LIN {X 0,Y 222.281,Z 512.285,A -85,B 0,C 180,E1 -22174.841,E2 -22174.841} C_VEL
LIN {X 0,Y 219.936,Z 524.701,A -85,B 0,C 180,E1 -22175.823,E2 -22175.823} C_VEL
LIN {X 0,Y 217.033,Z 536.462,A -85,B 0,C 180,E1 -22177.118,E2 -22177.118} C_VEL
LIN {X 0,Y 213.717,Z 547.223,A -85,B 0,C 180,E1 -22178.669,E2 -22178.669} C_VEL
LIN {X 0,Y 209.672,Z 558.118,A -85,B 0,C 180,E1 -22180.681,E2 -22180.681} C_VEL
LIN {X 0,Y 206.055,Z 566.605,A -85,B 0,C 180,E1 -22182.687,E2 -22182.687} C_VEL
LIN {X 0,Y 201.983,Z 575.031,A -85,B 0,C 180,E1 -22185.204,E2 -22185.204} C_VEL
LIN {X 0,Y 197.556,Z 583.105,A -85,B 0,C 180,E1 -22188.338,E2 -22188.338} C_VEL
LIN {X 0,Y 193.488,Z 589.856,A -85,B 0,C 180,E1 -22191.868,E2 -22191.868} C_VEL
LIN {X 0,Y 190.43,Z 594.406,A -85,B 0,C 180,E1 -22195.108,E2 -22195.108} C_VEL
LIN {X 0,Y 187.913,Z 597.772,A -85,B 0,C 180,E1 -22198.426,E2 -22198.426} C_VEL
LIN {X 0,Y 186.57,Z 599.41,A -85,B 0,C 180,E1 -22200.68,E2 -22200.68} C_VEL
LIN {X 0,Y 185.448,Z 600.607,A -85,B 0,C 180,E1 -22202.951,E2 -22202.951} C_VEL
LIN {X 0,Y 184.224,Z 601.526,A -85,B 0,C 180,E1 -22206.29,E2 -22206.29} C_VEL
LIN {X 0,Y 183.363,Z 601.506,A -85,B 0,C 180,E1 -22209.821,E2 -22209.821} C_VEL
LIN {X 0,Y 183.025,Z 600.3,A -85,B 0,C 180,E1 -22213.738,E2 -22213.738} C_VEL
LIN {X 0,Y 183.035,Z 598.555,A -85,B 0,C 180,E1 -22216.681,E2 -22216.681} C_VEL
LIN {X 0,Y 183.469,Z 595.61,A -85,B 0,C 180,E1 -22220.074,E2 -22220.074} C_VEL
LIN {X 0,Y 184.219,Z 591.613,A -85,B 0,C 180,E1 -22223.428,E2 -22223.428} C_VEL
LIN {X 0,Y 185.498,Z 585.472,A -85,B 0,C 180,E1 -22227.286,E2 -22227.286} C_VEL
LIN {X 0,Y 186.993,Z 578.75,A -85,B 0,C 180,E1 -22230.538,E2 -22230.538} C_VEL
LIN {X 0,Y 189.001,Z 570.397,A -85,B 0,C 180,E1 -22233.731,E2 -22233.731} C_VEL
LIN {X 0,Y 191.015,Z 561.82,A -85,B 0,C 180,E1 -22236.337,E2 -22236.337} C_VEL
LIN {X 0,Y 193.269,Z 551.234,A -85,B 0,C 180,E1 -22238.89,E2 -22238.89} C_VEL
LIN {X 0,Y 195.356,Z 540.725,A -85,B 0,C 180,E1 -22240.887,E2 -22240.887} C_VEL
LIN {X 0,Y 197.304,Z 529.166,A -85,B 0,C 180,E1 -22242.601,E2 -22242.601} C_VEL
LIN {X 0,Y 198.932,Z 517.169,A -85,B 0,C 180,E1 -22243.926,E2 -22243.926} C_VEL
LIN {X 0,Y 200.159,Z 504.209,A -85,B 0,C 180,E1 -22244.947,E2 -22244.947} C_VEL
LIN {X 0,Y 200.893,Z 491.969,A -85,B 0,C 180,E1 -22245.549,E2 -22245.549} C_VEL
LIN {X 0,Y 203.334,Z 436.009,A -85,B 0,C 180,E1 -22247.426,E2 -22247.426} C_VEL
LIN {X 0,Y 199.401,Z 426.13,A -85,B 0,C 180,E1 -22248.427,E2 -22248.427} C_VEL
LIN {X 0,Y 192.691,Z 412.029,A -85,B 0,C 180,E1 -22250.125,E2 -22250.125} C_VEL
LIN {X 0,Y 186.668,Z 401.306,A -85,B 0,C 180,E1 -22251.692,E2 -22251.692} C_VEL
LIN {X 0,Y 185.603,Z 398.365,A -85,B 0,C 180,E1 -22252.033,E2 -22252.033} C_VEL
LIN {X 0,Y 185.566,Z 398.373,A -85,B 0,C 180,E1 -22257.031,E2 -22257.031} C_VEL
LIN {X 0,Y 185.581,Z 398.368,A -85,B 0,C 180,E1 -22259.492,E2 -22259.492} C_VEL
LIN {X 0,Y 185.501,Z 398.379,A -85,B 0,C 180,E1 -22264.631,E2 -22264.631} C_VEL
LIN {X 0,Y 185.506,Z 398.373,A -85,B 0,C 180,E1 -22267.312,E2 -22267.312} C_VEL
LIN {X 0,Y 185.472,Z 398.376,A -85,B 0,C 180,E1 -22270.724,E2 -22270.724} C_VEL
LIN {X 0,Y 185.461,Z 398.376,A -85,B 0,C 180,E1 -22276.053,E2 -22276.053} C_VEL
LIN {X 0,Y 185.468,Z 398.38,A -85,B 0,C 180,E1 -22279.894,E2 -22279.894} C_VEL
LIN {X 0,Y 185.505,Z 398.369,A -85,B 0,C 180,E1 -22282.71,E2 -22282.71} C_VEL
LIN {X 0,Y 185.541,Z 398.369,A -85,B 0,C 180,E1 -22287.974,E2 -22287.974} C_VEL
LIN {X 0,Y 185.58,Z 398.361,A -85,B 0,C 180,E1 -22290.575,E2 -22290.575} C_VEL
LIN {X 0,Y 185.585,Z 398.36,A -85,B 0,C 180,E1 -22295.381,E2 -22295.381} C_VEL
LIN {X 0,Y 185.672,Z 398.353,A -85,B 0,C 180,E1 -22301.132,E2 -22301.132} C_VEL
LIN {X 0,Y 185.692,Z 398.345,A -85,B 0,C 180,E1 -22304.636,E2 -22304.636} C_VEL
LIN {X 0,Y 185.886,Z 398.322,A -85,B 0,C 180,E1 -22309.417,E2 -22309.417} C_VEL
LIN {X 0,Y 185.948,Z 398.319,A -85,B 0,C 180,E1 -22313.489,E2 -22313.489} C_VEL
LIN {X 0,Y 186.203,Z 398.276,A -85,B 0,C 180,E1 -22317.836,E2 -22317.836} C_VEL
LIN {X 0,Y 186.402,Z 398.23,A -85,B 0,C 180,E1 -22319.999,E2 -22319.999} C_VEL
LIN {X 0,Y 185.914,Z 398.307,A -85,B 0,C 180,E1 -22324.335,E2 -22324.335} C_VEL
LIN {X 0,Y 185.979,Z 398.318,A -85,B 0,C 180,E1 -22328.693,E2 -22328.693} C_VEL
LIN {X 0,Y 185.725,Z 398.347,A -85,B 0,C 180,E1 -22333.123,E2 -22333.123} C_VEL
LIN {X 0,Y 185.686,Z 398.349,A -85,B 0,C 180,E1 -22337.625,E2 -22337.625} C_VEL
LIN {X 0,Y 185.593,Z 398.365,A -85,B 0,C 180,E1 -22342.251,E2 -22342.251} C_VEL
LIN {X 0,Y 185.559,Z 398.369,A -85,B 0,C 180,E1 -22347.032,E2 -22347.032} C_VEL
LIN {X 0,Y 185.576,Z 398.37,A -85,B 0,C 180,E1 -22349.493,E2 -22349.493} C_VEL
LIN {X 0,Y 185.518,Z 398.38,A -85,B 0,C 180,E1 -22354.628,E2 -22354.628} C_VEL
LIN {X 0,Y 185.565,Z 398.375,A -85,B 0,C 180,E1 -22357.314,E2 -22357.314} C_VEL
LIN {X 0,Y 185.559,Z 398.377,A -85,B 0,C 180,E1 -22360.758,E2 -22360.758} C_VEL
LIN {X 0,Y 185.562,Z 398.375,A -85,B 0,C 180,E1 -22366.022,E2 -22366.022} C_VEL
LIN {X 0,Y 185.597,Z 398.469,A -85,B 0,C 180,E1 -22368.091,E2 -22368.091} C_VEL
LIN {X 0,Y 187.363,Z 405.749,A -85,B 0,C 180,E1 -22371.972,E2 -22371.972} C_VEL
LIN {X 0,Y 193.883,Z 421.299,A -85,B 0,C 180,E1 -22373.81,E2 -22373.81} C_VEL
LIN {X 0,Y 199.191,Z 435.84,A -85,B 0,C 180,E1 -22375.277,E2 -22375.277} C_VEL
LIN {X 0,Y 202.246,Z 467.615,A -85,B 0,C 180,E1 -22377.009,E2 -22377.009} C_VEL
LIN {X 0,Y 201.243,Z 492.996,A -85,B 0,C 180,E1 -22377.874,E2 -22377.874} C_VEL
LIN {X 0,Y 200.356,Z 498.833,A -85,B 0,C 180,E1 -22377.976,E2 -22377.976} C_VEL
LIN {X 0,Y 194.089,Z 517.66,A -85,B 0,C 180,E1 -22377.992,E2 -22377.992} C_VEL
LIN {X 0,Y 193.08,Z 523.397,A -85,B 0,C 180,E1 -22378.283,E2 -22378.283} C_VEL
LIN {X 0,Y 191.502,Z 536.392,A -85,B 0,C 180,E1 -22379.39,E2 -22379.39} C_VEL
LIN {X 0,Y 189.488,Z 548.643,A -85,B 0,C 180,E1 -22380.87,E2 -22380.87} C_VEL
LIN {X 0,Y 187.158,Z 559.674,A -85,B 0,C 180,E1 -22382.613,E2 -22382.613} C_VEL
LIN {X 0,Y 184.678,Z 570.968,A -85,B 0,C 180,E1 -22384.953,E2 -22384.953} C_VEL
LIN {X 0,Y 182.546,Z 580.085,A -85,B 0,C 180,E1 -22387.357,E2 -22387.357} C_VEL
LIN {X 0,Y 181.162,Z 585.57,A -85,B 0,C 180,E1 -22389.077,E2 -22389.077} C_VEL
LIN {X 0,Y 179.534,Z 592.745,A -85,B 0,C 180,E1 -22391.75,E2 -22391.75} C_VEL
LIN {X 0,Y 177.925,Z 600.065,A -85,B 0,C 180,E1 -22395.123,E2 -22395.123} C_VEL
LIN {X 0,Y 176.898,Z 605.891,A -85,B 0,C 180,E1 -22398.542,E2 -22398.542} C_VEL
LIN {X 0,Y 176.379,Z 610.455,A -85,B 0,C 180,E1 -22401.984,E2 -22401.984} C_VEL
LIN {X 0,Y 176.174,Z 614.18,A -85,B 0,C 180,E1 -22405.792,E2 -22405.792} C_VEL
LIN {X 0,Y 176.394,Z 616.866,A -85,B 0,C 180,E1 -22410,E2 -22410} C_VEL
LIN {X 0,Y 176.156,Z 618.092,A -85,B 0,C 180,E1 -22414.128,E2 -22414.128} C_VEL
LIN {X 0,Y 176.21,Z 618.167,A -85,B 0,C 180,E1 -22416.872,E2 -22416.872} C_VEL
LIN {X 0,Y 176.95,Z 617.068,A -85,B 0,C 180,E1 -22421.454,E2 -22421.454} C_VEL
LIN {X 0,Y 177.682,Z 615.947,A -85,B 0,C 180,E1 -22423.728,E2 -22423.728} C_VEL
LIN {X 0,Y 178.687,Z 614.389,A -85,B 0,C 180,E1 -22425.981,E2 -22425.981} C_VEL
LIN {X 0,Y 180.91,Z 611.301,A -85,B 0,C 180,E1 -22429.281,E2 -22429.281} C_VEL
LIN {X 0,Y 183.636,Z 607.189,A -85,B 0,C 180,E1 -22432.501,E2 -22432.501} C_VEL
LIN {X 0,Y 187.434,Z 600.937,A -85,B 0,C 180,E1 -22436.139,E2 -22436.139} C_VEL
LIN {X 0,Y 191.356,Z 594.172,A -85,B 0,C 180,E1 -22439.119,E2 -22439.119} C_VEL
LIN {X 0,Y 195.968,Z 585.811,A -85,B 0,C 180,E1 -22441.936,E2 -22441.936} C_VEL
LIN {X 0,Y 200.127,Z 577.24,A -85,B 0,C 180,E1 -22444.185,E2 -22444.185} C_VEL
LIN {X 0,Y 204.678,Z 566.714,A -85,B 0,C 180,E1 -22446.32,E2 -22446.32} C_VEL
LIN {X 0,Y 208.619,Z 556.305,A -85,B 0,C 180,E1 -22447.937,E2 -22447.937} C_VEL
LIN {X 0,Y 212.179,Z 544.891,A -85,B 0,C 180,E1 -22449.306,E2 -22449.306} C_VEL
LIN {X 0,Y 215.33,Z 531.845,A -85,B 0,C 180,E1 -22450.441,E2 -22450.441} C_VEL
LIN {X 0,Y 217.654,Z 518.383,A -85,B 0,C 180,E1 -22451.247,E2 -22451.247} C_VEL
LIN {X 0,Y 218.894,Z 505.408,A -85,B 0,C 180,E1 -22451.736,E2 -22451.736} C_VEL
LIN {X 0,Y 220.857,Z 474.587,A -85,B 0,C 180,E1 -22452.675,E2 -22452.675} C_VEL
LIN {X 0,Y 220.319,Z 470.267,A -85,B 0,C 180,E1 -22453.05,E2 -22453.05} C_VEL
LIN {X 0,Y 215.13,Z 457.835,A -85,B 0,C 180,E1 -22455.335,E2 -22455.335} C_VEL
LIN {X 0,Y 209.768,Z 446.74,A -85,B 0,C 180,E1 -22457.874,E2 -22457.874} C_VEL
LIN {X 0,Y 204.194,Z 436.795,A -85,B 0,C 180,E1 -22460.756,E2 -22460.756} C_VEL
LIN {X 0,Y 201.189,Z 431.731,A -85,B 0,C 180,E1 -22462.459,E2 -22462.459} C_VEL
LIN {X 0,Y 197.894,Z 426.511,A -85,B 0,C 180,E1 -22464.466,E2 -22464.466} C_VEL
LIN {X 0,Y 194.017,Z 420.666,A -85,B 0,C 180,E1 -22467.088,E2 -22467.088} C_VEL
LIN {X 0,Y 190.602,Z 415.814,A -85,B 0,C 180,E1 -22469.73,E2 -22469.73} C_VEL
LIN {X 0,Y 189.536,Z 414.282,A -85,B 0,C 180,E1 -22470.639,E2 -22470.639} C_VEL
LIN {X 0,Y 185.502,Z 408.804,A -85,B 0,C 180,E1 -22474.537,E2 -22474.537} C_VEL
LIN {X 0,Y 184.714,Z 407.543,A -85,B 0,C 180,E1 -22475.441,E2 -22475.441} C_VEL
LIN {X 0,Y 181.501,Z 404.142,A -85,B 0,C 180,E1 -22479.605,E2 -22479.605} C_VEL
LIN {X 0,Y 179.041,Z 400.824,A -85,B 0,C 180,E1 -22484.49,E2 -22484.49} C_VEL
LIN {X 0,Y 178.646,Z 399.226,A -85,B 0,C 180,E1 -22486.202,E2 -22486.202} C_VEL
LIN {X 0,Y 178.955,Z 399.184,A -85,B 0,C 180,E1 -22490.963,E2 -22490.963} C_VEL
LIN {X 0,Y 179.15,Z 399.152,A -85,B 0,C 180,E1 -22497.752,E2 -22497.752} C_VEL
LIN {X 0,Y 179.315,Z 399.229,A -85,B 0,C 180,E1 -22500.351,E2 -22500.351} C_VEL
LIN {X 0,Y 179.788,Z 401.258,A -85,B 0,C 180,E1 -22501.821,E2 -22501.821} C_VEL
LIN {X 0,Y 181.116,Z 403.543,A -85,B 0,C 180,E1 -22504.452,E2 -22504.452} C_VEL
LIN {X 0,Y 184.311,Z 405.474,A -85,B 0,C 180,E1 -22508.567,E2 -22508.567} C_VEL
LIN {X 0,Y 185.791,Z 408.533,A -85,B 0,C 180,E1 -22510.377,E2 -22510.377} C_VEL
LIN {X 0,Y 188.224,Z 410.668,A -85,B 0,C 180,E1 -22512.672,E2 -22512.672} C_VEL
LIN {X 0,Y 188.96,Z 411.267,A -85,B 0,C 180,E1 -22513.306,E2 -22513.306} C_VEL
LIN {X 0,Y 190.801,Z 414.301,A -85,B 0,C 180,E1 -22514.943,E2 -22514.943} C_VEL
LIN {X 0,Y 193.337,Z 416.734,A -85,B 0,C 180,E1 -22516.839,E2 -22516.839} C_VEL
LIN {X 0,Y 195.579,Z 420.044,A -85,B 0,C 180,E1 -22518.465,E2 -22518.465} C_VEL
LIN {X 0,Y 197.368,Z 422.01,A -85,B 0,C 180,E1 -22519.604,E2 -22519.604} C_VEL
LIN {X 0,Y 200.297,Z 425.823,A -85,B 0,C 180,E1 -22521.385,E2 -22521.385} C_VEL
LIN {X 0,Y 204.844,Z 432.293,A -85,B 0,C 180,E1 -22523.921,E2 -22523.921} C_VEL
LIN {X 0,Y 209.465,Z 439.033,A -85,B 0,C 180,E1 -22526.238,E2 -22526.238} C_VEL
LIN {X 0,Y 215.672,Z 449.023,A -85,B 0,C 180,E1 -22529.062,E2 -22529.062} C_VEL
LIN {X 0,Y 219.882,Z 456.772,A -85,B 0,C 180,E1 -22530.825,E2 -22530.825} C_VEL
LIN {X 0,Y 221.735,Z 460.811,A -85,B 0,C 180,E1 -22531.591,E2 -22531.591} C_VEL
LIN {X 0,Y 219.07,Z 499.801,A -85,B 0,C 180,E1 -22532.809,E2 -22532.809} C_VEL
LIN {X 0,Y 217.235,Z 513.449,A -85,B 0,C 180,E1 -22533.56,E2 -22533.56} C_VEL
LIN {X 0,Y 214.826,Z 525.527,A -85,B 0,C 180,E1 -22534.54,E2 -22534.54} C_VEL
LIN {X 0,Y 211.585,Z 537.865,A -85,B 0,C 180,E1 -22535.941,E2 -22535.941} C_VEL
LIN {X 0,Y 207.934,Z 549.072,A -85,B 0,C 180,E1 -22537.626,E2 -22537.626} C_VEL
LIN {X 0,Y 203.941,Z 559.145,A -85,B 0,C 180,E1 -22539.552,E2 -22539.552} C_VEL
LIN {X 0,Y 199.411,Z 569.061,A -85,B 0,C 180,E1 -22542.04,E2 -22542.04} C_VEL
LIN {X 0,Y 195.133,Z 577.215,A -85,B 0,C 180,E1 -22544.659,E2 -22544.659} C_VEL
LIN {X 0,Y 190.814,Z 584.63,A -85,B 0,C 180,E1 -22547.758,E2 -22547.758} C_VEL
LIN {X 0,Y 187.617,Z 589.599,A -85,B 0,C 180,E1 -22550.447,E2 -22550.447} C_VEL
LIN {X 0,Y 184.211,Z 594.421,A -85,B 0,C 180,E1 -22553.872,E2 -22553.872} C_VEL
LIN {X 0,Y 181.551,Z 597.797,A -85,B 0,C 180,E1 -22557.184,E2 -22557.184} C_VEL
LIN {X 0,Y 180.078,Z 599.495,A -85,B 0,C 180,E1 -22559.513,E2 -22559.513} C_VEL
LIN {X 0,Y 178.792,Z 600.76,A -85,B 0,C 180,E1 -22561.856,E2 -22561.856} C_VEL
LIN {X 0,Y 177.277,Z 601.87,A -85,B 0,C 180,E1 -22565.76,E2 -22565.76} C_VEL
LIN {X 0,Y 176.405,Z 601.882,A -85,B 0,C 180,E1 -22568.989,E2 -22568.989} C_VEL
LIN {X 0,Y 176.063,Z 601.421,A -85,B 0,C 180,E1 -22571.377,E2 -22571.377} C_VEL
LIN {X 0,Y 175.949,Z 600.495,A -85,B 0,C 180,E1 -22573.764,E2 -22573.764} C_VEL
LIN {X 0,Y 175.927,Z 599.158,A -85,B 0,C 180,E1 -22576.132,E2 -22576.132} C_VEL
LIN {X 0,Y 176.282,Z 596.333,A -85,B 0,C 180,E1 -22579.665,E2 -22579.665} C_VEL
LIN {X 0,Y 177.051,Z 592.457,A -85,B 0,C 180,E1 -22583.161,E2 -22583.161} C_VEL
LIN {X 0,Y 178.082,Z 587.45,A -85,B 0,C 180,E1 -22586.606,E2 -22586.606} C_VEL
LIN {X 0,Y 179.517,Z 581.158,A -85,B 0,C 180,E1 -22590,E2 -22590} C_VEL
LIN {X 0,Y 181.476,Z 573.284,A -85,B 0,C 180,E1 -22593.33,E2 -22593.33} C_VEL
LIN {X 0,Y 183.442,Z 565.238,A -85,B 0,C 180,E1 -22596.048,E2 -22596.048} C_VEL
LIN {X 0,Y 185.817,Z 555.399,A -85,B 0,C 180,E1 -22598.701,E2 -22598.701} C_VEL
LIN {X 0,Y 187.782,Z 545.805,A -85,B 0,C 180,E1 -22600.785,E2 -22600.785} C_VEL
LIN {X 0,Y 189.817,Z 535.446,A -85,B 0,C 180,E1 -22602.563,E2 -22602.563} C_VEL
LIN {X 0,Y 191.722,Z 523.136,A -85,B 0,C 180,E1 -22604.19,E2 -22604.19} C_VEL
LIN {X 0,Y 193.209,Z 510.227,A -85,B 0,C 180,E1 -22605.426,E2 -22605.426} C_VEL
LIN {X 0,Y 194.24,Z 497.73,A -85,B 0,C 180,E1 -22606.217,E2 -22606.217} C_VEL
LIN {X 0,Y 197.004,Z 437.596,A -85,B 0,C 180,E1 -22608.331,E2 -22608.331} C_VEL
LIN {X 0,Y 191.815,Z 425.138,A -85,B 0,C 180,E1 -22609.712,E2 -22609.712} C_VEL
LIN {X 0,Y 185.069,Z 411.727,A -85,B 0,C 180,E1 -22611.523,E2 -22611.523} C_VEL
LIN {X 0,Y 179.955,Z 402.686,A -85,B 0,C 180,E1 -22612.96,E2 -22612.96} C_VEL
LIN {X 0,Y 178.668,Z 400,A -85,B 0,C 180,E1 -22613.357,E2 -22613.357} C_VEL
LIN {X 0,Y 178.523,Z 399.234,A -85,B 0,C 180,E1 -22613.484,E2 -22613.484} C_VEL
LIN {X 0,Y 178.49,Z 399.251,A -85,B 0,C 180,E1 -22618.196,E2 -22618.196} C_VEL
LIN {X 0,Y 178.503,Z 399.253,A -85,B 0,C 180,E1 -22620.785,E2 -22620.785} C_VEL
LIN {X 0,Y 178.487,Z 399.252,A -85,B 0,C 180,E1 -22624.218,E2 -22624.218} C_VEL
LIN {X 0,Y 178.396,Z 399.264,A -85,B 0,C 180,E1 -22629.073,E2 -22629.073} C_VEL
LIN {X 0,Y 178.399,Z 399.255,A -85,B 0,C 180,E1 -22632.044,E2 -22632.044} C_VEL
LIN {X 0,Y 178.395,Z 399.259,A -85,B 0,C 180,E1 -22635.162,E2 -22635.162} C_VEL
LIN {X 0,Y 178.403,Z 399.257,A -85,B 0,C 180,E1 -22638.458,E2 -22638.458} C_VEL
LIN {X 0,Y 178.421,Z 399.254,A -85,B 0,C 180,E1 -22643.782,E2 -22643.782} C_VEL
LIN {X 0,Y 178.484,Z 399.253,A -85,B 0,C 180,E1 -22646.545,E2 -22646.545} C_VEL
LIN {X 0,Y 178.521,Z 399.239,A -85,B 0,C 180,E1 -22650.006,E2 -22650.006} C_VEL
LIN {X 0,Y 178.523,Z 399.241,A -85,B 0,C 180,E1 -22654.882,E2 -22654.882} C_VEL
LIN {X 0,Y 178.621,Z 399.233,A -85,B 0,C 180,E1 -22660.783,E2 -22660.783} C_VEL
LIN {X 0,Y 178.654,Z 399.228,A -85,B 0,C 180,E1 -22666.347,E2 -22666.347} C_VEL
LIN {X 0,Y 178.911,Z 399.187,A -85,B 0,C 180,E1 -22670.959,E2 -22670.959} C_VEL
LIN {X 0,Y 178.866,Z 399.201,A -85,B 0,C 180,E1 -22675.492,E2 -22675.492} C_VEL
LIN {X 0,Y 179.366,Z 399.105,A -85,B 0,C 180,E1 -22679.999,E2 -22679.999} C_VEL
LIN {X 0,Y 178.862,Z 399.185,A -85,B 0,C 180,E1 -22684.507,E2 -22684.507} C_VEL
LIN {X 0,Y 178.907,Z 399.198,A -85,B 0,C 180,E1 -22689.04,E2 -22689.04} C_VEL
LIN {X 0,Y 178.653,Z 399.228,A -85,B 0,C 180,E1 -22693.652,E2 -22693.652} C_VEL
LIN {X 0,Y 178.62,Z 399.232,A -85,B 0,C 180,E1 -22699.216,E2 -22699.216} C_VEL
LIN {X 0,Y 178.531,Z 399.246,A -85,B 0,C 180,E1 -22705.124,E2 -22705.124} C_VEL
LIN {X 0,Y 178.476,Z 399.255,A -85,B 0,C 180,E1 -22710.791,E2 -22710.791} C_VEL
LIN {X 0,Y 178.482,Z 399.258,A -85,B 0,C 180,E1 -22714.22,E2 -22714.22} C_VEL
LIN {X 0,Y 178.47,Z 399.26,A -85,B 0,C 180,E1 -22719.055,E2 -22719.055} C_VEL
LIN {X 0,Y 178.497,Z 399.258,A -85,B 0,C 180,E1 -22722.016,E2 -22722.016} C_VEL
LIN {X 0,Y 178.529,Z 399.317,A -85,B 0,C 180,E1 -22727.116,E2 -22727.116} C_VEL
LIN {X 0,Y 180.026,Z 405.349,A -85,B 0,C 180,E1 -22730.522,E2 -22730.522} C_VEL
LIN {X 0,Y 187.418,Z 422.385,A -85,B 0,C 180,E1 -22732.724,E2 -22732.724} C_VEL
LIN {X 0,Y 193.121,Z 437.955,A -85,B 0,C 180,E1 -22734.391,E2 -22734.391} C_VEL
LIN {X 0,Y 195.928,Z 467.915,A -85,B 0,C 180,E1 -22736.091,E2 -22736.091} C_VEL
LIN {X 0,Y 193.825,Z 514.316,A -85,B 0,C 180,E1 -22737.745,E2 -22737.745} C_VEL
LIN {X 0,Y 193.08,Z 523.397,A -85,B 0,C 180,E1 -22738.283,E2 -22738.283} C_VEL
LIN {X 0,Y 191.912,Z 529.074,A -85,B 0,C 180,E1 -22738.622,E2 -22738.622} C_VEL
LIN {X 0,Y 188.076,Z 538.074,A -85,B 0,C 180,E1 -22739.117,E2 -22739.117} C_VEL
LIN {X 0,Y 183.906,Z 546.775,A -85,B 0,C 180,E1 -22739.846,E2 -22739.846} C_VEL
LIN {X 0,Y 182.235,Z 551.985,A -85,B 0,C 180,E1 -22740.551,E2 -22740.551} C_VEL
LIN {X 0,Y 179.822,Z 562.227,A -85,B 0,C 180,E1 -22742.348,E2 -22742.348} C_VEL
LIN {X 0,Y 177.947,Z 570.778,A -85,B 0,C 180,E1 -22744.251,E2 -22744.251} C_VEL
LIN {X 0,Y 175.612,Z 580.306,A -85,B 0,C 180,E1 -22746.872,E2 -22746.872} C_VEL
LIN {X 0,Y 174.172,Z 585.886,A -85,B 0,C 180,E1 -22748.706,E2 -22748.706} C_VEL
LIN {X 0,Y 172.171,Z 594.492,A -85,B 0,C 180,E1 -22752.173,E2 -22752.173} C_VEL
LIN {X 0,Y 170.54,Z 601.357,A -85,B 0,C 180,E1 -22755.685,E2 -22755.685} C_VEL
LIN {X 0,Y 169.653,Z 606.846,A -85,B 0,C 180,E1 -22759.257,E2 -22759.257} C_VEL
LIN {X 0,Y 169.237,Z 611.11,A -85,B 0,C 180,E1 -22762.844,E2 -22762.844} C_VEL
LIN {X 0,Y 169.088,Z 613.927,A -85,B 0,C 180,E1 -22765.978,E2 -22765.978} C_VEL
LIN {X 0,Y 169.31,Z 616.411,A -85,B 0,C 180,E1 -22770,E2 -22770} C_VEL
LIN {X 0,Y 169.078,Z 617.648,A -85,B 0,C 180,E1 -22773.976,E2 -22773.976} C_VEL
LIN {X 0,Y 169.139,Z 617.848,A -85,B 0,C 180,E1 -22777.161,E2 -22777.161} C_VEL
LIN {X 0,Y 169.976,Z 616.818,A -85,B 0,C 180,E1 -22781.931,E2 -22781.931} C_VEL
LIN {X 0,Y 170.747,Z 615.737,A -85,B 0,C 180,E1 -22784.297,E2 -22784.297} C_VEL
LIN {X 0,Y 171.852,Z 614.247,A -85,B 0,C 180,E1 -22786.634,E2 -22786.634} C_VEL
LIN {X 0,Y 174.207,Z 611.227,A -85,B 0,C 180,E1 -22790.054,E2 -22790.054} C_VEL
LIN {X 0,Y 177.093,Z 607.188,A -85,B 0,C 180,E1 -22793.381,E2 -22793.381} C_VEL
LIN {X 0,Y 181.079,Z 601.037,A -85,B 0,C 180,E1 -22797.13,E2 -22797.13} C_VEL
LIN {X 0,Y 185.181,Z 594.375,A -85,B 0,C 180,E1 -22800.189,E2 -22800.189} C_VEL
LIN {X 0,Y 190.003,Z 586.143,A -85,B 0,C 180,E1 -22803.064,E2 -22803.064} C_VEL
LIN {X 0,Y 194.327,Z 577.753,A -85,B 0,C 180,E1 -22805.355,E2 -22805.355} C_VEL
LIN {X 0,Y 199.035,Z 567.432,A -85,B 0,C 180,E1 -22807.524,E2 -22807.524} C_VEL
LIN {X 0,Y 203.627,Z 555.83,A -85,B 0,C 180,E1 -22809.359,E2 -22809.359} C_VEL
LIN {X 0,Y 207.332,Z 544.367,A -85,B 0,C 180,E1 -22810.731,E2 -22810.731} C_VEL
LIN {X 0,Y 210.583,Z 531.259,A -85,B 0,C 180,E1 -22811.872,E2 -22811.872} C_VEL
LIN {X 0,Y 212.824,Z 518.755,A -85,B 0,C 180,E1 -22812.625,E2 -22812.625} C_VEL
LIN {X 0,Y 214.188,Z 505.476,A -85,B 0,C 180,E1 -22813.141,E2 -22813.141} C_VEL
LIN {X 0,Y 216.16,Z 475.771,A -85,B 0,C 180,E1 -22814.055,E2 -22814.055} C_VEL
LIN {X 0,Y 215.814,Z 473.339,A -85,B 0,C 180,E1 -22814.292,E2 -22814.292} C_VEL
LIN {X 0,Y 210.516,Z 460.485,A -85,B 0,C 180,E1 -22816.799,E2 -22816.799} C_VEL
LIN {X 0,Y 206.06,Z 451.173,A -85,B 0,C 180,E1 -22819.062,E2 -22819.062} C_VEL
LIN {X 0,Y 200.931,Z 441.751,A -85,B 0,C 180,E1 -22821.891,E2 -22821.891} C_VEL
LIN {X 0,Y 198.036,Z 436.799,A -85,B 0,C 180,E1 -22823.637,E2 -22823.637} C_VEL
LIN {X 0,Y 195.352,Z 432.363,A -85,B 0,C 180,E1 -22825.379,E2 -22825.379} C_VEL
LIN {X 0,Y 191.747,Z 426.753,A -85,B 0,C 180,E1 -22827.974,E2 -22827.974} C_VEL
LIN {X 0,Y 188.425,Z 421.719,A -85,B 0,C 180,E1 -22830.723,E2 -22830.723} C_VEL
LIN {X 0,Y 183.755,Z 415.061,A -85,B 0,C 180,E1 -22835.422,E2 -22835.422} C_VEL
LIN {X 0,Y 183.077,Z 414.113,A -85,B 0,C 180,E1 -22836.23,E2 -22836.23} C_VEL
LIN {X 0,Y 180.321,Z 411.049,A -85,B 0,C 180,E1 -22839.999,E2 -22839.999} C_VEL
LIN {X 0,Y 177.97,Z 407.679,A -85,B 0,C 180,E1 -22844.981,E2 -22844.981} C_VEL
LIN {X 0,Y 177.643,Z 406.407,A -85,B 0,C 180,E1 -22846.269,E2 -22846.269} C_VEL
LIN {X 0,Y 176.717,Z 405.923,A -85,B 0,C 180,E1 -22853.836,E2 -22853.836} C_VEL
LIN {X 0,Y 178.184,Z 406.278,A -85,B 0,C 180,E1 -22859.789,E2 -22859.789} C_VEL
LIN {X 0,Y 179.233,Z 409.428,A -85,B 0,C 180,E1 -22862.669,E2 -22862.669} C_VEL
LIN {X 0,Y 181.153,Z 411.342,A -85,B 0,C 180,E1 -22865.846,E2 -22865.846} C_VEL
LIN {X 0,Y 182.823,Z 412.312,A -85,B 0,C 180,E1 -22867.941,E2 -22867.941} C_VEL
LIN {X 0,Y 184.47,Z 415.457,A -85,B 0,C 180,E1 -22869.994,E2 -22869.994} C_VEL
LIN {X 0,Y 187.244,Z 418.031,A -85,B 0,C 180,E1 -22872.671,E2 -22872.671} C_VEL
LIN {X 0,Y 189.583,Z 421.46,A -85,B 0,C 180,E1 -22874.766,E2 -22874.766} C_VEL
LIN {X 0,Y 191.414,Z 423.378,A -85,B 0,C 180,E1 -22876.19,E2 -22876.19} C_VEL
LIN {X 0,Y 194.135,Z 427.088,A -85,B 0,C 180,E1 -22878.2,E2 -22878.2} C_VEL
LIN {X 0,Y 195.455,Z 428.858,A -85,B 0,C 180,E1 -22879.094,E2 -22879.094} C_VEL
LIN {X 0,Y 198.831,Z 433.445,A -85,B 0,C 180,E1 -22881.207,E2 -22881.207} C_VEL
LIN {X 0,Y 202.172,Z 438.26,A -85,B 0,C 180,E1 -22883.128,E2 -22883.128} C_VEL
LIN {X 0,Y 207.098,Z 445.716,A -85,B 0,C 180,E1 -22885.706,E2 -22885.706} C_VEL
LIN {X 0,Y 212.47,Z 454.636,A -85,B 0,C 180,E1 -22888.258,E2 -22888.258} C_VEL
LIN {X 0,Y 216.254,Z 461.842,A -85,B 0,C 180,E1 -22889.936,E2 -22889.936} C_VEL
LIN {X 0,Y 217.007,Z 463.534,A -85,B 0,C 180,E1 -22890.267,E2 -22890.267} C_VEL
LIN {X 0,Y 214.352,Z 500.142,A -85,B 0,C 180,E1 -22891.409,E2 -22891.409} C_VEL
LIN {X 0,Y 212.485,Z 513.593,A -85,B 0,C 180,E1 -22892.153,E2 -22892.153} C_VEL
LIN {X 0,Y 209.907,Z 526.081,A -85,B 0,C 180,E1 -22893.173,E2 -22893.173} C_VEL
LIN {X 0,Y 206.762,Z 537.633,A -85,B 0,C 180,E1 -22894.487,E2 -22894.487} C_VEL
LIN {X 0,Y 202.807,Z 549.333,A -85,B 0,C 180,E1 -22896.248,E2 -22896.248} C_VEL
LIN {X 0,Y 198.788,Z 559.109,A -85,B 0,C 180,E1 -22898.13,E2 -22898.13} C_VEL
LIN {X 0,Y 194.205,Z 568.75,A -85,B 0,C 180,E1 -22900.541,E2 -22900.541} C_VEL
LIN {X 0,Y 189.939,Z 576.596,A -85,B 0,C 180,E1 -22903.05,E2 -22903.05} C_VEL
LIN {X 0,Y 185.559,Z 583.825,A -85,B 0,C 180,E1 -22906.024,E2 -22906.024} C_VEL
LIN {X 0,Y 181.855,Z 589.291,A -85,B 0,C 180,E1 -22908.931,E2 -22908.931} C_VEL
LIN {X 0,Y 178.799,Z 593.495,A -85,B 0,C 180,E1 -22911.827,E2 -22911.827} C_VEL
LIN {X 0,Y 175.283,Z 597.791,A -85,B 0,C 180,E1 -22915.853,E2 -22915.853} C_VEL
LIN {X 0,Y 173.655,Z 599.581,A -85,B 0,C 180,E1 -22918.257,E2 -22918.257} C_VEL
LIN {X 0,Y 172.216,Z 600.906,A -85,B 0,C 180,E1 -22920.679,E2 -22920.679} C_VEL
LIN {X 0,Y 170.325,Z 602.217,A -85,B 0,C 180,E1 -22925.201,E2 -22925.201} C_VEL
LIN {X 0,Y 169.501,Z 602.257,A -85,B 0,C 180,E1 -22928.09,E2 -22928.09} C_VEL
LIN {X 0,Y 169.07,Z 601.855,A -85,B 0,C 180,E1 -22930.577,E2 -22930.577} C_VEL
LIN {X 0,Y 168.839,Z 600.967,A -85,B 0,C 180,E1 -22933.216,E2 -22933.216} C_VEL
LIN {X 0,Y 168.823,Z 599.757,A -85,B 0,C 180,E1 -22935.536,E2 -22935.536} C_VEL
LIN {X 0,Y 169.122,Z 597.048,A -85,B 0,C 180,E1 -22939.222,E2 -22939.222} C_VEL
LIN {X 0,Y 169.904,Z 593.012,A -85,B 0,C 180,E1 -22943.104,E2 -22943.104} C_VEL
LIN {X 0,Y 170.909,Z 588.415,A -85,B 0,C 180,E1 -22946.464,E2 -22946.464} C_VEL
LIN {X 0,Y 172.34,Z 582.269,A -85,B 0,C 180,E1 -22950,E2 -22950} C_VEL
LIN {X 0,Y 174.323,Z 574.619,A -85,B 0,C 180,E1 -22953.467,E2 -22953.467} C_VEL
LIN {X 0,Y 176.345,Z 566.793,A -85,B 0,C 180,E1 -22956.292,E2 -22956.292} C_VEL
LIN {X 0,Y 178.777,Z 557.208,A -85,B 0,C 180,E1 -22959.047,E2 -22959.047} C_VEL
LIN {X 0,Y 181.078,Z 546.617,A -85,B 0,C 180,E1 -22961.473,E2 -22961.473} C_VEL
LIN {X 0,Y 183.46,Z 534.744,A -85,B 0,C 180,E1 -22963.57,E2 -22963.57} C_VEL
LIN {X 0,Y 185.476,Z 522.051,A -85,B 0,C 180,E1 -22965.24,E2 -22965.24} C_VEL
LIN {X 0,Y 186.973,Z 509.401,A -85,B 0,C 180,E1 -22966.444,E2 -22966.444} C_VEL
LIN {X 0,Y 187.938,Z 497.425,A -85,B 0,C 180,E1 -22967.197,E2 -22967.197} C_VEL
LIN {X 0,Y 190.698,Z 439.225,A -85,B 0,C 180,E1 -22969.294,E2 -22969.294} C_VEL
LIN {X 0,Y 184.672,Z 425.186,A -85,B 0,C 180,E1 -22970.987,E2 -22970.987} C_VEL
LIN {X 0,Y 177.199,Z 410.848,A -85,B 0,C 180,E1 -22973.143,E2 -22973.143} C_VEL
LIN {X 0,Y 172.846,Z 403.443,A -85,B 0,C 180,E1 -22974.456,E2 -22974.456} C_VEL
LIN {X 0,Y 171.562,Z 400.569,A -85,B 0,C 180,E1 -22974.895,E2 -22974.895} C_VEL
LIN {X 0,Y 171.499,Z 400.11,A -85,B 0,C 180,E1 -22975,E2 -22975} C_VEL
LIN {X 0,Y 171.461,Z 400.13,A -85,B 0,C 180,E1 -22980.595,E2 -22980.595} C_VEL
LIN {X 0,Y 171.394,Z 400.136,A -85,B 0,C 180,E1 -22985.033,E2 -22985.033} C_VEL
LIN {X 0,Y 171.358,Z 400.139,A -85,B 0,C 180,E1 -22988.806,E2 -22988.806} C_VEL
LIN {X 0,Y 171.322,Z 400.142,A -85,B 0,C 180,E1 -22994.216,E2 -22994.216} C_VEL
LIN {X 0,Y 171.335,Z 400.14,A -85,B 0,C 180,E1 -22998.98,E2 -22998.98} C_VEL
LIN {X 0,Y 171.386,Z 400.128,A -85,B 0,C 180,E1 -23002.04,E2 -23002.04} C_VEL
LIN {X 0,Y 171.397,Z 400.134,A -85,B 0,C 180,E1 -23005.091,E2 -23005.091} C_VEL
LIN {X 0,Y 171.447,Z 400.121,A -85,B 0,C 180,E1 -23010.533,E2 -23010.533} C_VEL
LIN {X 0,Y 171.451,Z 400.118,A -85,B 0,C 180,E1 -23015.8,E2 -23015.8} C_VEL
LIN {X 0,Y 171.577,Z 400.11,A -85,B 0,C 180,E1 -23020.871,E2 -23020.871} C_VEL
LIN {X 0,Y 171.572,Z 400.108,A -85,B 0,C 180,E1 -23025.772,E2 -23025.772} C_VEL
LIN {X 0,Y 171.847,Z 400.067,A -85,B 0,C 180,E1 -23030.584,E2 -23030.584} C_VEL
LIN {X 0,Y 171.814,Z 400.079,A -85,B 0,C 180,E1 -23035.307,E2 -23035.307} C_VEL
LIN {X 0,Y 172.328,Z 399.979,A -85,B 0,C 180,E1 -23039.999,E2 -23039.999} C_VEL
LIN {X 0,Y 171.81,Z 400.064,A -85,B 0,C 180,E1 -23044.692,E2 -23044.692} C_VEL
LIN {X 0,Y 171.844,Z 400.077,A -85,B 0,C 180,E1 -23049.415,E2 -23049.415} C_VEL
LIN {X 0,Y 171.571,Z 400.112,A -85,B 0,C 180,E1 -23054.227,E2 -23054.227} C_VEL
LIN {X 0,Y 171.541,Z 400.114,A -85,B 0,C 180,E1 -23059.561,E2 -23059.561} C_VEL
LIN {X 0,Y 171.466,Z 400.127,A -85,B 0,C 180,E1 -23065.617,E2 -23065.617} C_VEL
LIN {X 0,Y 171.439,Z 400.132,A -85,B 0,C 180,E1 -23070.587,E2 -23070.587} C_VEL
LIN {X 0,Y 171.401,Z 400.138,A -85,B 0,C 180,E1 -23075.032,E2 -23075.032} C_VEL
LIN {X 0,Y 171.425,Z 400.139,A -85,B 0,C 180,E1 -23078.837,E2 -23078.837} C_VEL
LIN {X 0,Y 171.44,Z 400.135,A -85,B 0,C 180,E1 -23084.178,E2 -23084.178} C_VEL
LIN {X 0,Y 171.479,Z 400.238,A -85,B 0,C 180,E1 -23086.1,E2 -23086.1} C_VEL
LIN {X 0,Y 172.681,Z 404.938,A -85,B 0,C 180,E1 -23088.919,E2 -23088.919} C_VEL
LIN {X 0,Y 179.928,Z 420.911,A -85,B 0,C 180,E1 -23091.236,E2 -23091.236} C_VEL
LIN {X 0,Y 186.601,Z 438.762,A -85,B 0,C 180,E1 -23093.307,E2 -23093.307} C_VEL
LIN {X 0,Y 187.25,Z 441.951,A -85,B 0,C 180,E1 -23093.563,E2 -23093.563} C_VEL
LIN {X 0,Y 189.61,Z 469.351,A -85,B 0,C 180,E1 -23095.158,E2 -23095.158} C_VEL
LIN {X 0,Y 187.51,Z 513.385,A -85,B 0,C 180,E1 -23096.76,E2 -23096.76} C_VEL
LIN {X 0,Y 186.255,Z 526.891,A -85,B 0,C 180,E1 -23097.634,E2 -23097.634} C_VEL
LIN {X 0,Y 184.454,Z 539.754,A -85,B 0,C 180,E1 -23098.886,E2 -23098.886} C_VEL
LIN {X 0,Y 182.235,Z 551.985,A -85,B 0,C 180,E1 -23100.551,E2 -23100.551} C_VEL
LIN {X 0,Y 180.531,Z 557.172,A -85,B 0,C 180,E1 -23101.342,E2 -23101.342} C_VEL
LIN {X 0,Y 176.039,Z 565.152,A -85,B 0,C 180,E1 -23102.596,E2 -23102.596} C_VEL
LIN {X 0,Y 171.473,Z 572.615,A -85,B 0,C 180,E1 -23104.097,E2 -23104.097} C_VEL
LIN {X 0,Y 169.681,Z 576.977,A -85,B 0,C 180,E1 -23105.253,E2 -23105.253} C_VEL
LIN {X 0,Y 167.43,Z 584.82,A -85,B 0,C 180,E1 -23107.804,E2 -23107.804} C_VEL
LIN {X 0,Y 165.998,Z 590.887,A -85,B 0,C 180,E1 -23110.203,E2 -23110.203} C_VEL
LIN {X 0,Y 164.152,Z 598.42,A -85,B 0,C 180,E1 -23113.842,E2 -23113.842} C_VEL
LIN {X 0,Y 162.892,Z 604.45,A -85,B 0,C 180,E1 -23117.542,E2 -23117.542} C_VEL
LIN {X 0,Y 162.276,Z 609.197,A -85,B 0,C 180,E1 -23121.282,E2 -23121.282} C_VEL
LIN {X 0,Y 162.018,Z 612.784,A -85,B 0,C 180,E1 -23125.023,E2 -23125.023} C_VEL
LIN {X 0,Y 162.055,Z 614.605,A -85,B 0,C 180,E1 -23127.514,E2 -23127.514} C_VEL
LIN {X 0,Y 162.227,Z 615.956,A -85,B 0,C 180,E1 -23130,E2 -23130} C_VEL
LIN {X 0,Y 161.996,Z 617.199,A -85,B 0,C 180,E1 -23133.784,E2 -23133.784} C_VEL
LIN {X 0,Y 162.074,Z 617.527,A -85,B 0,C 180,E1 -23137.475,E2 -23137.475} C_VEL
LIN {X 0,Y 162.987,Z 616.568,A -85,B 0,C 180,E1 -23142.45,E2 -23142.45} C_VEL
LIN {X 0,Y 165.047,Z 614.092,A -85,B 0,C 180,E1 -23147.341,E2 -23147.341} C_VEL
LIN {X 0,Y 167.523,Z 611.131,A -85,B 0,C 180,E1 -23150.891,E2 -23150.891} C_VEL
LIN {X 0,Y 171.365,Z 606.094,A -85,B 0,C 180,E1 -23155.112,E2 -23155.112} C_VEL
LIN {X 0,Y 175.451,Z 600.144,A -85,B 0,C 180,E1 -23158.729,E2 -23158.729} C_VEL
LIN {X 0,Y 179.875,Z 593.362,A -85,B 0,C 180,E1 -23161.834,E2 -23161.834} C_VEL
LIN {X 0,Y 184.948,Z 584.975,A -85,B 0,C 180,E1 -23164.749,E2 -23164.749} C_VEL
LIN {X 0,Y 189.57,Z 576.371,A -85,B 0,C 180,E1 -23167.044,E2 -23167.044} C_VEL
LIN {X 0,Y 194.526,Z 565.812,A -85,B 0,C 180,E1 -23169.215,E2 -23169.215} C_VEL
LIN {X 0,Y 198.776,Z 555.354,A -85,B 0,C 180,E1 -23170.85,E2 -23170.85} C_VEL
LIN {X 0,Y 202.604,Z 543.844,A -85,B 0,C 180,E1 -23172.227,E2 -23172.227} C_VEL
LIN {X 0,Y 205.734,Z 531.78,A -85,B 0,C 180,E1 -23173.284,E2 -23173.284} C_VEL
LIN {X 0,Y 208.122,Z 519.065,A -85,B 0,C 180,E1 -23174.072,E2 -23174.072} C_VEL
LIN {X 0,Y 209.565,Z 506.24,A -85,B 0,C 180,E1 -23174.588,E2 -23174.588} C_VEL
LIN {X 0,Y 211.598,Z 476.949,A -85,B 0,C 180,E1 -23175.494,E2 -23175.494} C_VEL
LIN {X 0,Y 206.551,Z 464.349,A -85,B 0,C 180,E1 -23178.067,E2 -23178.067} C_VEL
LIN {X 0,Y 202.348,Z 455.44,A -85,B 0,C 180,E1 -23180.347,E2 -23180.347} C_VEL
LIN {X 0,Y 197.959,Z 447.114,A -85,B 0,C 180,E1 -23182.931,E2 -23182.931} C_VEL
LIN {X 0,Y 195.173,Z 442.201,A -85,B 0,C 180,E1 -23184.717,E2 -23184.717} C_VEL
LIN {X 0,Y 192.738,Z 438.089,A -85,B 0,C 180,E1 -23186.396,E2 -23186.396} C_VEL
LIN {X 0,Y 189.558,Z 432.872,A -85,B 0,C 180,E1 -23188.857,E2 -23188.857} C_VEL
LIN {X 0,Y 185.768,Z 426.987,A -85,B 0,C 180,E1 -23192.238,E2 -23192.238} C_VEL
LIN {X 0,Y 182.161,Z 421.563,A -85,B 0,C 180,E1 -23196.178,E2 -23196.178} C_VEL
LIN {X 0,Y 179.307,Z 418.06,A -85,B 0,C 180,E1 -23200.164,E2 -23200.164} C_VEL
LIN {X 0,Y 176.893,Z 414.471,A -85,B 0,C 180,E1 -23205.549,E2 -23205.549} C_VEL
LIN {X 0,Y 176.617,Z 413.291,A -85,B 0,C 180,E1 -23206.774,E2 -23206.774} C_VEL
LIN {X 0,Y 175.787,Z 412.945,A -85,B 0,C 180,E1 -23213.112,E2 -23213.112} C_VEL
LIN {X 0,Y 177.105,Z 413.276,A -85,B 0,C 180,E1 -23219.29,E2 -23219.29} C_VEL
LIN {X 0,Y 178.325,Z 416.664,A -85,B 0,C 180,E1 -23222.683,E2 -23222.683} C_VEL
LIN {X 0,Y 180.46,Z 418.552,A -85,B 0,C 180,E1 -23226.149,E2 -23226.149} C_VEL
LIN {X 0,Y 181.411,Z 419.229,A -85,B 0,C 180,E1 -23227.374,E2 -23227.374} C_VEL
LIN {X 0,Y 183.21,Z 422.425,A -85,B 0,C 180,E1 -23229.662,E2 -23229.662} C_VEL
LIN {X 0,Y 185.535,Z 424.652,A -85,B 0,C 180,E1 -23232,E2 -23232} C_VEL
LIN {X 0,Y 187.906,Z 428.092,A -85,B 0,C 180,E1 -23234.209,E2 -23234.209} C_VEL
LIN {X 0,Y 189.49,Z 429.888,A -85,B 0,C 180,E1 -23235.503,E2 -23235.503} C_VEL
LIN {X 0,Y 192.347,Z 433.745,A -85,B 0,C 180,E1 -23237.687,E2 -23237.687} C_VEL
LIN {X 0,Y 196.793,Z 440.14,A -85,B 0,C 180,E1 -23240.666,E2 -23240.666} C_VEL
LIN {X 0,Y 201.301,Z 446.811,A -85,B 0,C 180,E1 -23243.307,E2 -23243.307} C_VEL
LIN {X 0,Y 207.009,Z 456.092,A -85,B 0,C 180,E1 -23246.3,E2 -23246.3} C_VEL
LIN {X 0,Y 211.945,Z 465.383,A -85,B 0,C 180,E1 -23248.672,E2 -23248.672} C_VEL
LIN {X 0,Y 212.397,Z 466.33,A -85,B 0,C 180,E1 -23248.882,E2 -23248.882} C_VEL
LIN {X 0,Y 209.8,Z 500.274,A -85,B 0,C 180,E1 -23249.939,E2 -23249.939} C_VEL
LIN {X 0,Y 207.805,Z 514.157,A -85,B 0,C 180,E1 -23250.713,E2 -23250.713} C_VEL
LIN {X 0,Y 205.072,Z 526.756,A -85,B 0,C 180,E1 -23251.753,E2 -23251.753} C_VEL
LIN {X 0,Y 202.08,Z 537.402,A -85,B 0,C 180,E1 -23252.964,E2 -23252.964} C_VEL
LIN {X 0,Y 198.411,Z 547.983,A -85,B 0,C 180,E1 -23254.524,E2 -23254.524} C_VEL
LIN {X 0,Y 193.758,Z 559.061,A -85,B 0,C 180,E1 -23256.63,E2 -23256.63} C_VEL
LIN {X 0,Y 189.422,Z 567.933,A -85,B 0,C 180,E1 -23258.819,E2 -23258.819} C_VEL
LIN {X 0,Y 184.907,Z 575.984,A -85,B 0,C 180,E1 -23261.354,E2 -23261.354} C_VEL
LIN {X 0,Y 180.809,Z 582.539,A -85,B 0,C 180,E1 -23263.974,E2 -23263.974} C_VEL
LIN {X 0,Y 176.259,Z 588.999,A -85,B 0,C 180,E1 -23267.326,E2 -23267.326} C_VEL
LIN {X 0,Y 172.492,Z 593.889,A -85,B 0,C 180,E1 -23270.728,E2 -23270.728} C_VEL
LIN {X 0,Y 169.088,Z 597.76,A -85,B 0,C 180,E1 -23274.417,E2 -23274.417} C_VEL
LIN {X 0,Y 167.001,Z 599.918,A -85,B 0,C 180,E1 -23277.319,E2 -23277.319} C_VEL
LIN {X 0,Y 164.433,Z 602.011,A -85,B 0,C 180,E1 -23281.957,E2 -23281.957} C_VEL
LIN {X 0,Y 163.42,Z 602.56,A -85,B 0,C 180,E1 -23284.574,E2 -23284.574} C_VEL
LIN {X 0,Y 162.624,Z 602.633,A -85,B 0,C 180,E1 -23287.112,E2 -23287.112} C_VEL
LIN {X 0,Y 162.095,Z 602.288,A -85,B 0,C 180,E1 -23289.705,E2 -23289.705} C_VEL
LIN {X 0,Y 161.766,Z 601.307,A -85,B 0,C 180,E1 -23292.904,E2 -23292.904} C_VEL
LIN {X 0,Y 161.797,Z 598.723,A -85,B 0,C 180,E1 -23297.457,E2 -23297.457} C_VEL
LIN {X 0,Y 162.397,Z 595.44,A -85,B 0,C 180,E1 -23301.288,E2 -23301.288} C_VEL
LIN {X 0,Y 163.342,Z 591.078,A -85,B 0,C 180,E1 -23305.064,E2 -23305.064} C_VEL
LIN {X 0,Y 164.644,Z 585.523,A -85,B 0,C 180,E1 -23308.777,E2 -23308.777} C_VEL
LIN {X 0,Y 166.451,Z 578.588,A -85,B 0,C 180,E1 -23312.42,E2 -23312.42} C_VEL
LIN {X 0,Y 168.379,Z 571.502,A -85,B 0,C 180,E1 -23315.389,E2 -23315.389} C_VEL
LIN {X 0,Y 170.733,Z 562.68,A -85,B 0,C 180,E1 -23318.367,E2 -23318.367} C_VEL
LIN {X 0,Y 173.24,Z 552.392,A -85,B 0,C 180,E1 -23321.11,E2 -23321.11} C_VEL
LIN {X 0,Y 175.597,Z 541.915,A -85,B 0,C 180,E1 -23323.305,E2 -23323.305} C_VEL
LIN {X 0,Y 177.793,Z 530.422,A -85,B 0,C 180,E1 -23325.181,E2 -23325.181} C_VEL
LIN {X 0,Y 179.636,Z 518.518,A -85,B 0,C 180,E1 -23326.624,E2 -23326.624} C_VEL
LIN {X 0,Y 181.033,Z 505.756,A -85,B 0,C 180,E1 -23327.728,E2 -23327.728} C_VEL
LIN {X 0,Y 181.909,Z 493.001,A -85,B 0,C 180,E1 -23328.421,E2 -23328.421} C_VEL
LIN {X 0,Y 184.494,Z 440.92,A -85,B 0,C 180,E1 -23330.309,E2 -23330.309} C_VEL
LIN {X 0,Y 178.265,Z 426.826,A -85,B 0,C 180,E1 -23332.157,E2 -23332.157} C_VEL
LIN {X 0,Y 171.737,Z 414.389,A -85,B 0,C 180,E1 -23334.156,E2 -23334.156} C_VEL
LIN {X 0,Y 166.168,Z 404.837,A -85,B 0,C 180,E1 -23335.966,E2 -23335.966} C_VEL
LIN {X 0,Y 164.628,Z 402.171,A -85,B 0,C 180,E1 -23336.497,E2 -23336.497} C_VEL
LIN {X 0,Y 164.382,Z 401.01,A -85,B 0,C 180,E1 -23336.674,E2 -23336.674} C_VEL
LIN {X 0,Y 164.391,Z 401.008,A -85,B 0,C 180,E1 -23341.234,E2 -23341.234} C_VEL
LIN {X 0,Y 164.296,Z 401.013,A -85,B 0,C 180,E1 -23346.788,E2 -23346.788} C_VEL
LIN {X 0,Y 164.292,Z 401.017,A -85,B 0,C 180,E1 -23349.915,E2 -23349.915} C_VEL
LIN {X 0,Y 164.28,Z 401.019,A -85,B 0,C 180,E1 -23353.341,E2 -23353.341} C_VEL
LIN {X 0,Y 164.263,Z 401.013,A -85,B 0,C 180,E1 -23356.798,E2 -23356.798} C_VEL
LIN {X 0,Y 164.295,Z 401.018,A -85,B 0,C 180,E1 -23360.351,E2 -23360.351} C_VEL
LIN {X 0,Y 164.329,Z 401.01,A -85,B 0,C 180,E1 -23364.348,E2 -23364.348} C_VEL
LIN {X 0,Y 164.388,Z 400.997,A -85,B 0,C 180,E1 -23369.133,E2 -23369.133} C_VEL
LIN {X 0,Y 164.409,Z 401,A -85,B 0,C 180,E1 -23374.692,E2 -23374.692} C_VEL
LIN {X 0,Y 164.483,Z 400.995,A -85,B 0,C 180,E1 -23380.05,E2 -23380.05} C_VEL
LIN {X 0,Y 164.502,Z 400.987,A -85,B 0,C 180,E1 -23385.146,E2 -23385.146} C_VEL
LIN {X 0,Y 164.766,Z 400.949,A -85,B 0,C 180,E1 -23390.176,E2 -23390.176} C_VEL
LIN {X 0,Y 164.831,Z 400.946,A -85,B 0,C 180,E1 -23392.65,E2 -23392.65} C_VEL
LIN {X 0,Y 165.045,Z 400.911,A -85,B 0,C 180,E1 -23397.559,E2 -23397.559} C_VEL
LIN {X 0,Y 165.291,Z 400.854,A -85,B 0,C 180,E1 -23399.999,E2 -23399.999} C_VEL
LIN {X 0,Y 164.758,Z 400.943,A -85,B 0,C 180,E1 -23404.893,E2 -23404.893} C_VEL
LIN {X 0,Y 164.827,Z 400.951,A -85,B 0,C 180,E1 -23407.349,E2 -23407.349} C_VEL
LIN {X 0,Y 164.699,Z 400.96,A -85,B 0,C 180,E1 -23411.06,E2 -23411.06} C_VEL
LIN {X 0,Y 164.479,Z 400.99,A -85,B 0,C 180,E1 -23417.403,E2 -23417.403} C_VEL
LIN {X 0,Y 164.47,Z 400.995,A -85,B 0,C 180,E1 -23419.989,E2 -23419.989} C_VEL
LIN {X 0,Y 164.391,Z 401.01,A -85,B 0,C 180,E1 -23426.134,E2 -23426.134} C_VEL
LIN {X 0,Y 164.373,Z 401.011,A -85,B 0,C 180,E1 -23431.228,E2 -23431.228} C_VEL
LIN {X 0,Y 164.345,Z 401.018,A -85,B 0,C 180,E1 -23436.776,E2 -23436.776} C_VEL
LIN {X 0,Y 164.366,Z 401.018,A -85,B 0,C 180,E1 -23439.894,E2 -23439.894} C_VEL
LIN {X 0,Y 164.433,Z 401.105,A -85,B 0,C 180,E1 -23444.963,E2 -23444.963} C_VEL
LIN {X 0,Y 165.26,Z 404.43,A -85,B 0,C 180,E1 -23447.115,E2 -23447.115} C_VEL
LIN {X 0,Y 167.435,Z 408.86,A -85,B 0,C 180,E1 -23447.889,E2 -23447.889} C_VEL
LIN {X 0,Y 173.439,Z 422.009,A -85,B 0,C 180,E1 -23449.939,E2 -23449.939} C_VEL
LIN {X 0,Y 178.37,Z 434.605,A -85,B 0,C 180,E1 -23451.571,E2 -23451.571} C_VEL
LIN {X 0,Y 181.106,Z 442.627,A -85,B 0,C 180,E1 -23452.475,E2 -23452.475} C_VEL
LIN {X 0,Y 183.378,Z 469.727,A -85,B 0,C 180,E1 -23454.121,E2 -23454.121} C_VEL
LIN {X 0,Y 181.166,Z 513.705,A -85,B 0,C 180,E1 -23455.775,E2 -23455.775} C_VEL
LIN {X 0,Y 179.871,Z 526.956,A -85,B 0,C 180,E1 -23456.671,E2 -23456.671} C_VEL
LIN {X 0,Y 178.007,Z 539.716,A -85,B 0,C 180,E1 -23457.959,E2 -23457.959} C_VEL
LIN {X 0,Y 175.69,Z 551.926,A -85,B 0,C 180,E1 -23459.684,E2 -23459.684} C_VEL
LIN {X 0,Y 172.917,Z 563.378,A -85,B 0,C 180,E1 -23461.805,E2 -23461.805} C_VEL
LIN {X 0,Y 170.683,Z 572.753,A -85,B 0,C 180,E1 -23464.057,E2 -23464.057} C_VEL
LIN {X 0,Y 169.681,Z 576.977,A -85,B 0,C 180,E1 -23465.253,E2 -23465.253} C_VEL
LIN {X 0,Y 167.926,Z 581.249,A -85,B 0,C 180,E1 -23466.505,E2 -23466.505} C_VEL
LIN {X 0,Y 163.478,Z 587.712,A -85,B 0,C 180,E1 -23468.602,E2 -23468.602} C_VEL
LIN {X 0,Y 159.111,Z 593.542,A -85,B 0,C 180,E1 -23470.999,E2 -23470.999} C_VEL
LIN {X 0,Y 157.53,Z 596.826,A -85,B 0,C 180,E1 -23472.687,E2 -23472.687} C_VEL
LIN {X 0,Y 155.919,Z 603.716,A -85,B 0,C 180,E1 -23476.975,E2 -23476.975} C_VEL
LIN {X 0,Y 155.228,Z 608.55,A -85,B 0,C 180,E1 -23480.882,E2 -23480.882} C_VEL
LIN {X 0,Y 154.937,Z 612.217,A -85,B 0,C 180,E1 -23484.795,E2 -23484.795} C_VEL
LIN {X 0,Y 154.958,Z 614.096,A -85,B 0,C 180,E1 -23487.401,E2 -23487.401} C_VEL
LIN {X 0,Y 155.145,Z 615.5,A -85,B 0,C 180,E1 -23490,E2 -23490} C_VEL
LIN {X 0,Y 154.928,Z 616.745,A -85,B 0,C 180,E1 -23493.639,E2 -23493.639} C_VEL
LIN {X 0,Y 155.003,Z 617.185,A -85,B 0,C 180,E1 -23497.818,E2 -23497.818} C_VEL
LIN {X 0,Y 155.382,Z 616.953,A -85,B 0,C 180,E1 -23500.423,E2 -23500.423} C_VEL
LIN {X 0,Y 156.943,Z 615.311,A -85,B 0,C 180,E1 -23505.586,E2 -23505.586} C_VEL
LIN {X 0,Y 158.275,Z 613.922,A -85,B 0,C 180,E1 -23508.109,E2 -23508.109} C_VEL
LIN {X 0,Y 160.867,Z 611.036,A -85,B 0,C 180,E1 -23511.798,E2 -23511.798} C_VEL
LIN {X 0,Y 164.112,Z 607.157,A -85,B 0,C 180,E1 -23515.356,E2 -23515.356} C_VEL
LIN {X 0,Y 167.851,Z 602.188,A -85,B 0,C 180,E1 -23518.783,E2 -23518.783} C_VEL
LIN {X 0,Y 172.258,Z 595.982,A -85,B 0,C 180,E1 -23522.031,E2 -23522.031} C_VEL
LIN {X 0,Y 177.34,Z 588.295,A -85,B 0,C 180,E1 -23525.073,E2 -23525.073} C_VEL
LIN {X 0,Y 182.995,Z 578.684,A -85,B 0,C 180,E1 -23527.914,E2 -23527.914} C_VEL
LIN {X 0,Y 188.029,Z 568.81,A -85,B 0,C 180,E1 -23530.146,E2 -23530.146} C_VEL
LIN {X 0,Y 192.935,Z 557.732,A -85,B 0,C 180,E1 -23532.015,E2 -23532.015} C_VEL
LIN {X 0,Y 197.448,Z 545.177,A -85,B 0,C 180,E1 -23533.6,E2 -23533.6} C_VEL
LIN {X 0,Y 200.699,Z 533.647,A -85,B 0,C 180,E1 -23534.675,E2 -23534.675} C_VEL
LIN {X 0,Y 203.433,Z 520.303,A -85,B 0,C 180,E1 -23535.541,E2 -23535.541} C_VEL
LIN {X 0,Y 205.063,Z 507.472,A -85,B 0,C 180,E1 -23536.08,E2 -23536.08} C_VEL
LIN {X 0,Y 207.151,Z 479.581,A -85,B 0,C 180,E1 -23536.939,E2 -23536.939} C_VEL
LIN {X 0,Y 202.633,Z 468.114,A -85,B 0,C 180,E1 -23539.414,E2 -23539.414} C_VEL
LIN {X 0,Y 198.513,Z 459.131,A -85,B 0,C 180,E1 -23541.824,E2 -23541.824} C_VEL
LIN {X 0,Y 193.526,Z 449.515,A -85,B 0,C 180,E1 -23545.041,E2 -23545.041} C_VEL
LIN {X 0,Y 190.155,Z 443.643,A -85,B 0,C 180,E1 -23547.498,E2 -23547.498} C_VEL
LIN {X 0,Y 187.345,Z 438.878,A -85,B 0,C 180,E1 -23549.819,E2 -23549.819} C_VEL
LIN {X 0,Y 184.036,Z 433.474,A -85,B 0,C 180,E1 -23552.956,E2 -23552.956} C_VEL
LIN {X 0,Y 180.314,Z 427.603,A -85,B 0,C 180,E1 -23557.332,E2 -23557.332} C_VEL
LIN {X 0,Y 177.978,Z 424.801,A -85,B 0,C 180,E1 -23560.874,E2 -23560.874} C_VEL
LIN {X 0,Y 175.8,Z 421.138,A -85,B 0,C 180,E1 -23566.269,E2 -23566.269} C_VEL
LIN {X 0,Y 175.592,Z 420.28,A -85,B 0,C 180,E1 -23567.284,E2 -23567.284} C_VEL
LIN {X 0,Y 175.153,Z 420.092,A -85,B 0,C 180,E1 -23575.398,E2 -23575.398} C_VEL
LIN {X 0,Y 176.067,Z 420.254,A -85,B 0,C 180,E1 -23578.857,E2 -23578.857} C_VEL
LIN {X 0,Y 177.22,Z 423.567,A -85,B 0,C 180,E1 -23582.273,E2 -23582.273} C_VEL
LIN {X 0,Y 179.571,Z 425.624,A -85,B 0,C 180,E1 -23586.179,E2 -23586.179} C_VEL
LIN {X 0,Y 180.07,Z 426.155,A -85,B 0,C 180,E1 -23586.865,E2 -23586.865} C_VEL
LIN {X 0,Y 181.934,Z 429.358,A -85,B 0,C 180,E1 -23589.31,E2 -23589.31} C_VEL
LIN {X 0,Y 183.888,Z 431.33,A -85,B 0,C 180,E1 -23591.358,E2 -23591.358} C_VEL
LIN {X 0,Y 186.63,Z 435.179,A -85,B 0,C 180,E1 -23593.977,E2 -23593.977} C_VEL
LIN {X 0,Y 187.709,Z 436.592,A -85,B 0,C 180,E1 -23594.902,E2 -23594.902} C_VEL
LIN {X 0,Y 191.209,Z 441.538,A -85,B 0,C 180,E1 -23597.656,E2 -23597.656} C_VEL
LIN {X 0,Y 195.74,Z 448.137,A -85,B 0,C 180,E1 -23600.717,E2 -23600.717} C_VEL
LIN {X 0,Y 201.598,Z 457.582,A -85,B 0,C 180,E1 -23604.152,E2 -23604.152} C_VEL
LIN {X 0,Y 206.765,Z 466.971,A -85,B 0,C 180,E1 -23606.856,E2 -23606.856} C_VEL
LIN {X 0,Y 207.904,Z 469.162,A -85,B 0,C 180,E1 -23607.419,E2 -23607.419} C_VEL
LIN {X 0,Y 205.403,Z 500.596,A -85,B 0,C 180,E1 -23608.406,E2 -23608.406} C_VEL
LIN {X 0,Y 203.346,Z 514.399,A -85,B 0,C 180,E1 -23609.175,E2 -23609.175} C_VEL
LIN {X 0,Y 200.669,Z 526.44,A -85,B 0,C 180,E1 -23610.162,E2 -23610.162} C_VEL
LIN {X 0,Y 197.546,Z 537.228,A -85,B 0,C 180,E1 -23611.371,E2 -23611.371} C_VEL
LIN {X 0,Y 193.642,Z 548.145,A -85,B 0,C 180,E1 -23612.985,E2 -23612.985} C_VEL
LIN {X 0,Y 188.884,Z 559.034,A -85,B 0,C 180,E1 -23615.059,E2 -23615.059} C_VEL
LIN {X 0,Y 183.678,Z 569.102,A -85,B 0,C 180,E1 -23617.585,E2 -23617.585} C_VEL
LIN {X 0,Y 178.22,Z 578.194,A -85,B 0,C 180,E1 -23620.616,E2 -23620.616} C_VEL
LIN {X 0,Y 173.468,Z 585.185,A -85,B 0,C 180,E1 -23623.687,E2 -23623.687} C_VEL
LIN {X 0,Y 169.335,Z 590.579,A -85,B 0,C 180,E1 -23626.781,E2 -23626.781} C_VEL
LIN {X 0,Y 165.391,Z 595.293,A -85,B 0,C 180,E1 -23630.403,E2 -23630.403} C_VEL
LIN {X 0,Y 163.038,Z 597.732,A -85,B 0,C 180,E1 -23632.881,E2 -23632.881} C_VEL
LIN {X 0,Y 160.367,Z 600.298,A -85,B 0,C 180,E1 -23636.375,E2 -23636.375} C_VEL
LIN {X 0,Y 157.855,Z 602.219,A -85,B 0,C 180,E1 -23640.677,E2 -23640.677} C_VEL
LIN {X 0,Y 156.496,Z 602.909,A -85,B 0,C 180,E1 -23643.921,E2 -23643.921} C_VEL
LIN {X 0,Y 155.16,Z 602.719,A -85,B 0,C 180,E1 -23648.755,E2 -23648.755} C_VEL
LIN {X 0,Y 154.688,Z 601.639,A -85,B 0,C 180,E1 -23652.576,E2 -23652.576} C_VEL
LIN {X 0,Y 154.796,Z 598.442,A -85,B 0,C 180,E1 -23658.211,E2 -23658.211} C_VEL
LIN {X 0,Y 155.485,Z 594.93,A -85,B 0,C 180,E1 -23662.207,E2 -23662.207} C_VEL
LIN {X 0,Y 156.527,Z 590.326,A -85,B 0,C 180,E1 -23666.138,E2 -23666.138} C_VEL
LIN {X 0,Y 158.284,Z 583.353,A -85,B 0,C 180,E1 -23670.636,E2 -23670.636} C_VEL
LIN {X 0,Y 160.422,Z 575.788,A -85,B 0,C 180,E1 -23674.397,E2 -23674.397} C_VEL
LIN {X 0,Y 162.605,Z 568.069,A -85,B 0,C 180,E1 -23677.45,E2 -23677.45} C_VEL
LIN {X 0,Y 165.239,Z 558.66,A -85,B 0,C 180,E1 -23680.414,E2 -23680.414} C_VEL
LIN {X 0,Y 167.734,Z 548.229,A -85,B 0,C 180,E1 -23683.015,E2 -23683.015} C_VEL
LIN {X 0,Y 170.296,Z 536.613,A -85,B 0,C 180,E1 -23685.253,E2 -23685.253} C_VEL
LIN {X 0,Y 172.497,Z 524.358,A -85,B 0,C 180,E1 -23687.028,E2 -23687.028} C_VEL
LIN {X 0,Y 174.266,Z 510.778,A -85,B 0,C 180,E1 -23688.441,E2 -23688.441} C_VEL
LIN {X 0,Y 175.426,Z 497.993,A -85,B 0,C 180,E1 -23689.299,E2 -23689.299} C_VEL
LIN {X 0,Y 178.281,Z 442.734,A -85,B 0,C 180,E1 -23691.401,E2 -23691.401} C_VEL
LIN {X 0,Y 172.658,Z 429.973,A -85,B 0,C 180,E1 -23693.174,E2 -23693.174} C_VEL
LIN {X 0,Y 165.65,Z 416.557,A -85,B 0,C 180,E1 -23695.471,E2 -23695.471} C_VEL
LIN {X 0,Y 160.886,Z 408.664,A -85,B 0,C 180,E1 -23697.119,E2 -23697.119} C_VEL
LIN {X 0,Y 159.103,Z 405.781,A -85,B 0,C 180,E1 -23697.767,E2 -23697.767} C_VEL
LIN {X 0,Y 157.606,Z 403.218,A -85,B 0,C 180,E1 -23698.332,E2 -23698.332} C_VEL
LIN {X 0,Y 157.284,Z 401.891,A -85,B 0,C 180,E1 -23698.524,E2 -23698.524} C_VEL
LIN {X 0,Y 157.283,Z 401.889,A -85,B 0,C 180,E1 -23702.425,E2 -23702.425} C_VEL
LIN {X 0,Y 157.269,Z 401.889,A -85,B 0,C 180,E1 -23706.448,E2 -23706.448} C_VEL
LIN {X 0,Y 157.211,Z 401.893,A -85,B 0,C 180,E1 -23712.109,E2 -23712.109} C_VEL
LIN {X 0,Y 157.193,Z 401.896,A -85,B 0,C 180,E1 -23717.882,E2 -23717.882} C_VEL
LIN {X 0,Y 157.267,Z 401.886,A -85,B 0,C 180,E1 -23723.55,E2 -23723.55} C_VEL
LIN {X 0,Y 157.292,Z 401.886,A -85,B 0,C 180,E1 -23728.095,E2 -23728.095} C_VEL
LIN {X 0,Y 157.316,Z 401.888,A -85,B 0,C 180,E1 -23733.464,E2 -23733.464} C_VEL
LIN {X 0,Y 157.392,Z 401.878,A -85,B 0,C 180,E1 -23739.667,E2 -23739.667} C_VEL
LIN {X 0,Y 157.439,Z 401.861,A -85,B 0,C 180,E1 -23744.464,E2 -23744.464} C_VEL
LIN {X 0,Y 157.687,Z 401.832,A -85,B 0,C 180,E1 -23749.73,E2 -23749.73} C_VEL
LIN {X 0,Y 157.767,Z 401.824,A -85,B 0,C 180,E1 -23752.319,E2 -23752.319} C_VEL
LIN {X 0,Y 158.253,Z 401.729,A -85,B 0,C 180,E1 -23759.999,E2 -23759.999} C_VEL
LIN {X 0,Y 157.764,Z 401.831,A -85,B 0,C 180,E1 -23767.68,E2 -23767.68} C_VEL
LIN {X 0,Y 157.634,Z 401.839,A -85,B 0,C 180,E1 -23771.236,E2 -23771.236} C_VEL
LIN {X 0,Y 157.449,Z 401.872,A -85,B 0,C 180,E1 -23775.534,E2 -23775.534} C_VEL
LIN {X 0,Y 157.367,Z 401.883,A -85,B 0,C 180,E1 -23780.933,E2 -23780.933} C_VEL
LIN {X 0,Y 157.312,Z 401.889,A -85,B 0,C 180,E1 -23786.685,E2 -23786.685} C_VEL
LIN {X 0,Y 157.275,Z 401.894,A -85,B 0,C 180,E1 -23792.427,E2 -23792.427} C_VEL
LIN {X 0,Y 157.32,Z 401.892,A -85,B 0,C 180,E1 -23796.477,E2 -23796.477} C_VEL
LIN {X 0,Y 157.285,Z 401.901,A -85,B 0,C 180,E1 -23802.086,E2 -23802.086} C_VEL
LIN {X 0,Y 157.358,Z 402.02,A -85,B 0,C 180,E1 -23803.737,E2 -23803.737} C_VEL
LIN {X 0,Y 157.87,Z 404.06,A -85,B 0,C 180,E1 -23805.13,E2 -23805.13} C_VEL
LIN {X 0,Y 160.208,Z 408.583,A -85,B 0,C 180,E1 -23806.03,E2 -23806.03} C_VEL
LIN {X 0,Y 166.439,Z 421.628,A -85,B 0,C 180,E1 -23808.319,E2 -23808.319} C_VEL
LIN {X 0,Y 171.463,Z 434.067,A -85,B 0,C 180,E1 -23810.107,E2 -23810.107} C_VEL
LIN {X 0,Y 175.141,Z 444.749,A -85,B 0,C 180,E1 -23811.406,E2 -23811.406} C_VEL
LIN {X 0,Y 177.204,Z 469.932,A -85,B 0,C 180,E1 -23813.007,E2 -23813.007} C_VEL
LIN {X 0,Y 174.963,Z 512.947,A -85,B 0,C 180,E1 -23814.659,E2 -23814.659} C_VEL
LIN {X 0,Y 173.635,Z 526.245,A -85,B 0,C 180,E1 -23815.571,E2 -23815.571} C_VEL
LIN {X 0,Y 171.819,Z 538.548,A -85,B 0,C 180,E1 -23816.834,E2 -23816.834} C_VEL
LIN {X 0,Y 169.618,Z 550.115,A -85,B 0,C 180,E1 -23818.46,E2 -23818.46} C_VEL
LIN {X 0,Y 166.99,Z 560.604,A -85,B 0,C 180,E1 -23820.363,E2 -23820.363} C_VEL
LIN {X 0,Y 164.576,Z 570.394,A -85,B 0,C 180,E1 -23822.674,E2 -23822.674} C_VEL
LIN {X 0,Y 161.908,Z 580.351,A -85,B 0,C 180,E1 -23825.648,E2 -23825.648} C_VEL
LIN {X 0,Y 160.416,Z 585.427,A -85,B 0,C 180,E1 -23827.459,E2 -23827.459} C_VEL
LIN {X 0,Y 158.585,Z 592.712,A -85,B 0,C 180,E1 -23830.587,E2 -23830.587} C_VEL
LIN {X 0,Y 157.53,Z 596.826,A -85,B 0,C 180,E1 -23832.687,E2 -23832.687} C_VEL
LIN {X 0,Y 156.055,Z 599.938,A -85,B 0,C 180,E1 -23834.46,E2 -23834.46} C_VEL
LIN {X 0,Y 152.247,Z 604.408,A -85,B 0,C 180,E1 -23837.438,E2 -23837.438} C_VEL
LIN {X 0,Y 148.81,Z 608.172,A -85,B 0,C 180,E1 -23840.678,E2 -23840.678} C_VEL
LIN {X 0,Y 147.948,Z 610.185,A -85,B 0,C 180,E1 -23842.796,E2 -23842.796} C_VEL
LIN {X 0,Y 147.883,Z 613.565,A -85,B 0,C 180,E1 -23847.276,E2 -23847.276} C_VEL
LIN {X 0,Y 148.064,Z 615.04,A -85,B 0,C 180,E1 -23850,E2 -23850} C_VEL
LIN {X 0,Y 147.859,Z 616.231,A -85,B 0,C 180,E1 -23853.476,E2 -23853.476} C_VEL
LIN {X 0,Y 147.958,Z 616.831,A -85,B 0,C 180,E1 -23858.192,E2 -23858.192} C_VEL
LIN {X 0,Y 148.366,Z 616.661,A -85,B 0,C 180,E1 -23860.922,E2 -23860.922} C_VEL
LIN {X 0,Y 150.08,Z 615.101,A -85,B 0,C 180,E1 -23866.318,E2 -23866.318} C_VEL
LIN {X 0,Y 153.315,Z 612.006,A -85,B 0,C 180,E1 -23871.513,E2 -23871.513} C_VEL
LIN {X 0,Y 156.506,Z 608.54,A -85,B 0,C 180,E1 -23875.252,E2 -23875.252} C_VEL
LIN {X 0,Y 160.25,Z 604.031,A -85,B 0,C 180,E1 -23878.843,E2 -23878.843} C_VEL
LIN {X 0,Y 165.473,Z 597.274,A -85,B 0,C 180,E1 -23882.786,E2 -23882.786} C_VEL
LIN {X 0,Y 170.707,Z 589.96,A -85,B 0,C 180,E1 -23885.92,E2 -23885.92} C_VEL
LIN {X 0,Y 176.476,Z 580.929,A -85,B 0,C 180,E1 -23888.845,E2 -23888.845} C_VEL
LIN {X 0,Y 182.183,Z 570.552,A -85,B 0,C 180,E1 -23891.346,E2 -23891.346} C_VEL
LIN {X 0,Y 187.177,Z 560.016,A -85,B 0,C 180,E1 -23893.253,E2 -23893.253} C_VEL
LIN {X 0,Y 191.831,Z 548.264,A -85,B 0,C 180,E1 -23894.849,E2 -23894.849} C_VEL
LIN {X 0,Y 195.809,Z 535.305,A -85,B 0,C 180,E1 -23896.132,E2 -23896.132} C_VEL
LIN {X 0,Y 198.727,Z 522.431,A -85,B 0,C 180,E1 -23897.037,E2 -23897.037} C_VEL
LIN {X 0,Y 200.575,Z 510.19,A -85,B 0,C 180,E1 -23897.586,E2 -23897.586} C_VEL
LIN {X 0,Y 202.734,Z 482.007,A -85,B 0,C 180,E1 -23898.505,E2 -23898.505} C_VEL
LIN {X 0,Y 198.651,Z 471.462,A -85,B 0,C 180,E1 -23900.922,E2 -23900.922} C_VEL
LIN {X 0,Y 194.958,Z 463.278,A -85,B 0,C 180,E1 -23903.253,E2 -23903.253} C_VEL
LIN {X 0,Y 190.563,Z 454.58,A -85,B 0,C 180,E1 -23906.311,E2 -23906.311} C_VEL
LIN {X 0,Y 187.766,Z 449.462,A -85,B 0,C 180,E1 -23908.526,E2 -23908.526} C_VEL
LIN {X 0,Y 185.283,Z 445.058,A -85,B 0,C 180,E1 -23910.713,E2 -23910.713} C_VEL
LIN {X 0,Y 182.038,Z 439.505,A -85,B 0,C 180,E1 -23914.008,E2 -23914.008} C_VEL
LIN {X 0,Y 178.676,Z 434.046,A -85,B 0,C 180,E1 -23918.268,E2 -23918.268} C_VEL
LIN {X 0,Y 176.639,Z 431.505,A -85,B 0,C 180,E1 -23921.654,E2 -23921.654} C_VEL
LIN {X 0,Y 174.771,Z 427.936,A -85,B 0,C 180,E1 -23926.816,E2 -23926.816} C_VEL
LIN {X 0,Y 174.595,Z 427.289,A -85,B 0,C 180,E1 -23927.727,E2 -23927.727} C_VEL
LIN {X 0,Y 174.815,Z 427.155,A -85,B 0,C 180,E1 -23937.697,E2 -23937.697} C_VEL
LIN {X 0,Y 175.079,Z 427.509,A -85,B 0,C 180,E1 -23938.644,E2 -23938.644} C_VEL
LIN {X 0,Y 176.31,Z 430.756,A -85,B 0,C 180,E1 -23942.285,E2 -23942.285} C_VEL
LIN {X 0,Y 178.7,Z 432.965,A -85,B 0,C 180,E1 -23946.28,E2 -23946.28} C_VEL
LIN {X 0,Y 180.665,Z 436.289,A -85,B 0,C 180,E1 -23948.952,E2 -23948.952} C_VEL
LIN {X 0,Y 182.377,Z 438.186,A -85,B 0,C 180,E1 -23950.829,E2 -23950.829} C_VEL
LIN {X 0,Y 185.215,Z 442.06,A -85,B 0,C 180,E1 -23953.612,E2 -23953.612} C_VEL
LIN {X 0,Y 189.094,Z 447.85,A -85,B 0,C 180,E1 -23956.88,E2 -23956.88} C_VEL
LIN {X 0,Y 193.397,Z 454.394,A -85,B 0,C 180,E1 -23959.957,E2 -23959.957} C_VEL
LIN {X 0,Y 199.149,Z 463.955,A -85,B 0,C 180,E1 -23963.484,E2 -23963.484} C_VEL
LIN {X 0,Y 203.547,Z 472.384,A -85,B 0,C 180,E1 -23965.914,E2 -23965.914} C_VEL
LIN {X 0,Y 201.01,Z 502.1,A -85,B 0,C 180,E1 -23966.86,E2 -23966.86} C_VEL
LIN {X 0,Y 198.867,Z 515.632,A -85,B 0,C 180,E1 -23967.641,E2 -23967.641} C_VEL
LIN {X 0,Y 195.807,Z 528.279,A -85,B 0,C 180,E1 -23968.705,E2 -23968.705} C_VEL
LIN {X 0,Y 192.014,Z 540.4,A -85,B 0,C 180,E1 -23970.152,E2 -23970.152} C_VEL
LIN {X 0,Y 187.901,Z 550.981,A -85,B 0,C 180,E1 -23971.815,E2 -23971.815} C_VEL
LIN {X 0,Y 183.038,Z 561.205,A -85,B 0,C 180,E1 -23973.87,E2 -23973.87} C_VEL
LIN {X 0,Y 177.902,Z 570.519,A -85,B 0,C 180,E1 -23976.341,E2 -23976.341} C_VEL
LIN {X 0,Y 172.496,Z 579.019,A -85,B 0,C 180,E1 -23979.277,E2 -23979.277} C_VEL
LIN {X 0,Y 168.215,Z 584.978,A -85,B 0,C 180,E1 -23981.951,E2 -23981.951} C_VEL
LIN {X 0,Y 163.947,Z 590.292,A -85,B 0,C 180,E1 -23984.984,E2 -23984.984} C_VEL
LIN {X 0,Y 159.647,Z 595.152,A -85,B 0,C 180,E1 -23988.676,E2 -23988.676} C_VEL
LIN {X 0,Y 155.956,Z 598.793,A -85,B 0,C 180,E1 -23992.53,E2 -23992.53} C_VEL
LIN {X 0,Y 152.982,Z 601.323,A -85,B 0,C 180,E1 -23996.546,E2 -23996.546} C_VEL
LIN {X 0,Y 151.372,Z 602.428,A -85,B 0,C 180,E1 -23999.289,E2 -23999.289} C_VEL
LIN {X 0,Y 149.632,Z 603.253,A -85,B 0,C 180,E1 -24003.179,E2 -24003.179} C_VEL
LIN {X 0,Y 148.254,Z 603.151,A -85,B 0,C 180,E1 -24007.714,E2 -24007.714} C_VEL
LIN {X 0,Y 147.609,Z 601.965,A -85,B 0,C 180,E1 -24012.225,E2 -24012.225} C_VEL
LIN {X 0,Y 147.533,Z 600.019,A -85,B 0,C 180,E1 -24016.221,E2 -24016.221} C_VEL
LIN {X 0,Y 147.998,Z 596.971,A -85,B 0,C 180,E1 -24020.433,E2 -24020.433} C_VEL
LIN {X 0,Y 148.954,Z 592.856,A -85,B 0,C 180,E1 -24024.585,E2 -24024.585} C_VEL
LIN {X 0,Y 150.545,Z 586.55,A -85,B 0,C 180,E1 -24029.331,E2 -24029.331} C_VEL
LIN {X 0,Y 152.503,Z 579.69,A -85,B 0,C 180,E1 -24033.302,E2 -24033.302} C_VEL
LIN {X 0,Y 155.06,Z 571.144,A -85,B 0,C 180,E1 -24037.16,E2 -24037.16} C_VEL
LIN {X 0,Y 157.599,Z 562.341,A -85,B 0,C 180,E1 -24040.275,E2 -24040.275} C_VEL
LIN {X 0,Y 160.147,Z 552.702,A -85,B 0,C 180,E1 -24042.997,E2 -24042.997} C_VEL
LIN {X 0,Y 162.742,Z 542.144,A -85,B 0,C 180,E1 -24045.337,E2 -24045.337} C_VEL
LIN {X 0,Y 165.152,Z 530.494,A -85,B 0,C 180,E1 -24047.33,E2 -24047.33} C_VEL
LIN {X 0,Y 167.162,Z 518.388,A -85,B 0,C 180,E1 -24048.856,E2 -24048.856} C_VEL
LIN {X 0,Y 168.718,Z 505.265,A -85,B 0,C 180,E1 -24050.022,E2 -24050.022} C_VEL
LIN {X 0,Y 169.606,Z 492.447,A -85,B 0,C 180,E1 -24050.721,E2 -24050.721} C_VEL
LIN {X 0,Y 172.17,Z 444.59,A -85,B 0,C 180,E1 -24052.554,E2 -24052.554} C_VEL
LIN {X 0,Y 166.368,Z 431.535,A -85,B 0,C 180,E1 -24054.511,E2 -24054.511} C_VEL
LIN {X 0,Y 158.617,Z 417.073,A -85,B 0,C 180,E1 -24057.259,E2 -24057.259} C_VEL
LIN {X 0,Y 154.093,Z 409.914,A -85,B 0,C 180,E1 -24058.953,E2 -24058.953} C_VEL
LIN {X 0,Y 152.406,Z 407.06,A -85,B 0,C 180,E1 -24059.633,E2 -24059.633} C_VEL
LIN {X 0,Y 150.646,Z 404.458,A -85,B 0,C 180,E1 -24060.342,E2 -24060.342} C_VEL
LIN {X 0,Y 150.22,Z 402.776,A -85,B 0,C 180,E1 -24060.611,E2 -24060.611} C_VEL
LIN {X 0,Y 150.194,Z 402.777,A -85,B 0,C 180,E1 -24064.16,E2 -24064.16} C_VEL
LIN {X 0,Y 150.178,Z 402.772,A -85,B 0,C 180,E1 -24067.471,E2 -24067.471} C_VEL
LIN {X 0,Y 150.15,Z 402.771,A -85,B 0,C 180,E1 -24071.503,E2 -24071.503} C_VEL
LIN {X 0,Y 150.126,Z 402.778,A -85,B 0,C 180,E1 -24075.394,E2 -24075.394} C_VEL
LIN {X 0,Y 150.141,Z 402.779,A -85,B 0,C 180,E1 -24079.054,E2 -24079.054} C_VEL
LIN {X 0,Y 150.178,Z 402.767,A -85,B 0,C 180,E1 -24082.706,E2 -24082.706} C_VEL
LIN {X 0,Y 150.214,Z 402.77,A -85,B 0,C 180,E1 -24087.367,E2 -24087.367} C_VEL
LIN {X 0,Y 150.241,Z 402.771,A -85,B 0,C 180,E1 -24092.719,E2 -24092.719} C_VEL
LIN {X 0,Y 150.349,Z 402.756,A -85,B 0,C 180,E1 -24099.207,E2 -24099.207} C_VEL
LIN {X 0,Y 150.35,Z 402.742,A -85,B 0,C 180,E1 -24103.711,E2 -24103.711} C_VEL
LIN {X 0,Y 150.609,Z 402.716,A -85,B 0,C 180,E1 -24109.242,E2 -24109.242} C_VEL
LIN {X 0,Y 150.704,Z 402.702,A -85,B 0,C 180,E1 -24111.957,E2 -24111.957} C_VEL
LIN {X 0,Y 151.214,Z 402.603,A -85,B 0,C 180,E1 -24119.999,E2 -24119.999} C_VEL
LIN {X 0,Y 150.701,Z 402.712,A -85,B 0,C 180,E1 -24128.042,E2 -24128.042} C_VEL
LIN {X 0,Y 150.574,Z 402.718,A -85,B 0,C 180,E1 -24131.436,E2 -24131.436} C_VEL
LIN {X 0,Y 150.357,Z 402.752,A -85,B 0,C 180,E1 -24136.287,E2 -24136.287} C_VEL
LIN {X 0,Y 150.348,Z 402.757,A -85,B 0,C 180,E1 -24140.792,E2 -24140.792} C_VEL
LIN {X 0,Y 150.241,Z 402.768,A -85,B 0,C 180,E1 -24147.282,E2 -24147.282} C_VEL
LIN {X 0,Y 150.215,Z 402.774,A -85,B 0,C 180,E1 -24152.634,E2 -24152.634} C_VEL
LIN {X 0,Y 150.231,Z 402.779,A -85,B 0,C 180,E1 -24157.456,E2 -24157.456} C_VEL
LIN {X 0,Y 150.253,Z 402.833,A -85,B 0,C 180,E1 -24162.307,E2 -24162.307} C_VEL
LIN {X 0,Y 150.526,Z 403.857,A -85,B 0,C 180,E1 -24162.916,E2 -24162.916} C_VEL
LIN {X 0,Y 152.836,Z 408.106,A -85,B 0,C 180,E1 -24163.897,E2 -24163.897} C_VEL
LIN {X 0,Y 159.478,Z 421.285,A -85,B 0,C 180,E1 -24166.546,E2 -24166.546} C_VEL
LIN {X 0,Y 165.555,Z 436.031,A -85,B 0,C 180,E1 -24168.866,E2 -24168.866} C_VEL
LIN {X 0,Y 169.203,Z 446.581,A -85,B 0,C 180,E1 -24170.24,E2 -24170.24} C_VEL
LIN {X 0,Y 171.059,Z 469.8,A -85,B 0,C 180,E1 -24171.792,E2 -24171.792} C_VEL
LIN {X 0,Y 168.791,Z 512.58,A -85,B 0,C 180,E1 -24173.494,E2 -24173.494} C_VEL
LIN {X 0,Y 167.373,Z 526.201,A -85,B 0,C 180,E1 -24174.459,E2 -24174.459} C_VEL
LIN {X 0,Y 165.484,Z 538.433,A -85,B 0,C 180,E1 -24175.757,E2 -24175.757} C_VEL
LIN {X 0,Y 163.543,Z 548.174,A -85,B 0,C 180,E1 -24177.144,E2 -24177.144} C_VEL
LIN {X 0,Y 160.864,Z 559.045,A -85,B 0,C 180,E1 -24179.114,E2 -24179.114} C_VEL
LIN {X 0,Y 158.631,Z 567.927,A -85,B 0,C 180,E1 -24181.197,E2 -24181.197} C_VEL
LIN {X 0,Y 155.995,Z 577.386,A -85,B 0,C 180,E1 -24183.944,E2 -24183.944} C_VEL
LIN {X 0,Y 153.656,Z 584.811,A -85,B 0,C 180,E1 -24186.61,E2 -24186.61} C_VEL
LIN {X 0,Y 151.812,Z 591.759,A -85,B 0,C 180,E1 -24189.684,E2 -24189.684} C_VEL
LIN {X 0,Y 149.88,Z 599.01,A -85,B 0,C 180,E1 -24193.66,E2 -24193.66} C_VEL
LIN {X 0,Y 148.631,Z 604.767,A -85,B 0,C 180,E1 -24197.715,E2 -24197.715} C_VEL
LIN {X 0,Y 148.038,Z 609.283,A -85,B 0,C 180,E1 -24201.812,E2 -24201.812} C_VEL
LIN {X 0,Y 147.948,Z 610.185,A -85,B 0,C 180,E1 -24202.796,E2 -24202.796} C_VEL
LIN {X 0,Y 147.551,Z 611.416,A -85,B 0,C 180,E1 -24204.24,E2 -24204.24} C_VEL
LIN {X 0,Y 146.138,Z 612.934,A -85,B 0,C 180,E1 -24206.411,E2 -24206.411} C_VEL
LIN {X 0,Y 141.822,Z 615.266,A -85,B 0,C 180,E1 -24211.655,E2 -24211.655} C_VEL
LIN {X 0,Y 140.805,Z 615.911,A -85,B 0,C 180,E1 -24214.052,E2 -24214.052} C_VEL
LIN {X 0,Y 140.727,Z 616.046,A -85,B 0,C 180,E1 -24214.867,E2 -24214.867} C_VEL
LIN {X 0,Y 140.911,Z 616.476,A -85,B 0,C 180,E1 -24218.605,E2 -24218.605} C_VEL
LIN {X 0,Y 142.154,Z 615.827,A -85,B 0,C 180,E1 -24224.311,E2 -24224.311} C_VEL
LIN {X 0,Y 143.247,Z 614.892,A -85,B 0,C 180,E1 -24227.119,E2 -24227.119} C_VEL
LIN {X 0,Y 146.69,Z 611.873,A -85,B 0,C 180,E1 -24232.537,E2 -24232.537} C_VEL
LIN {X 0,Y 150.107,Z 608.493,A -85,B 0,C 180,E1 -24236.409,E2 -24236.409} C_VEL
LIN {X 0,Y 154.066,Z 604.077,A -85,B 0,C 180,E1 -24240.117,E2 -24240.117} C_VEL
LIN {X 0,Y 158.713,Z 598.508,A -85,B 0,C 180,E1 -24243.608,E2 -24243.608} C_VEL
LIN {X 0,Y 164.058,Z 591.599,A -85,B 0,C 180,E1 -24246.85,E2 -24246.85} C_VEL
LIN {X 0,Y 169.99,Z 582.991,A -85,B 0,C 180,E1 -24249.852,E2 -24249.852} C_VEL
LIN {X 0,Y 175.305,Z 574.204,A -85,B 0,C 180,E1 -24252.182,E2 -24252.182} C_VEL
LIN {X 0,Y 179.8,Z 565.756,A -85,B 0,C 180,E1 -24253.931,E2 -24253.931} C_VEL
LIN {X 0,Y 185.112,Z 554.098,A -85,B 0,C 180,E1 -24255.774,E2 -24255.774} C_VEL
LIN {X 0,Y 189.353,Z 542.514,A -85,B 0,C 180,E1 -24257.14,E2 -24257.14} C_VEL
LIN {X 0,Y 192.952,Z 529.78,A -85,B 0,C 180,E1 -24258.224,E2 -24258.224} C_VEL
LIN {X 0,Y 195.482,Z 517.545,A -85,B 0,C 180,E1 -24258.933,E2 -24258.933} C_VEL
LIN {X 0,Y 197.05,Z 504.139,A -85,B 0,C 180,E1 -24259.468,E2 -24259.468} C_VEL
LIN {X 0,Y 198.559,Z 484.752,A -85,B 0,C 180,E1 -24260.081,E2 -24260.081} C_VEL
LIN {X 0,Y 194.897,Z 474.989,A -85,B 0,C 180,E1 -24262.437,E2 -24262.437} C_VEL
LIN {X 0,Y 190.449,Z 465.114,A -85,B 0,C 180,E1 -24265.516,E2 -24265.516} C_VEL
LIN {X 0,Y 186.379,Z 456.823,A -85,B 0,C 180,E1 -24268.777,E2 -24268.777} C_VEL
LIN {X 0,Y 183.309,Z 451.271,A -85,B 0,C 180,E1 -24271.589,E2 -24271.589} C_VEL
LIN {X 0,Y 180.304,Z 445.882,A -85,B 0,C 180,E1 -24274.843,E2 -24274.843} C_VEL
LIN {X 0,Y 177.293,Z 440.759,A -85,B 0,C 180,E1 -24278.914,E2 -24278.914} C_VEL
LIN {X 0,Y 175.624,Z 438.512,A -85,B 0,C 180,E1 -24281.858,E2 -24281.858} C_VEL
LIN {X 0,Y 173.782,Z 434.952,A -85,B 0,C 180,E1 -24287.167,E2 -24287.167} C_VEL
LIN {X 0,Y 173.572,Z 434.282,A -85,B 0,C 180,E1 -24288.32,E2 -24288.32} C_VEL
LIN {X 0,Y 174.007,Z 434.238,A -85,B 0,C 180,E1 -24297.975,E2 -24297.975} C_VEL
LIN {X 0,Y 175.14,Z 437.539,A -85,B 0,C 180,E1 -24301.715,E2 -24301.715} C_VEL
LIN {X 0,Y 177.367,Z 439.745,A -85,B 0,C 180,E1 -24305.686,E2 -24305.686} C_VEL
LIN {X 0,Y 179.407,Z 443.188,A -85,B 0,C 180,E1 -24308.59,E2 -24308.59} C_VEL
LIN {X 0,Y 180.706,Z 444.689,A -85,B 0,C 180,E1 -24310.08,E2 -24310.08} C_VEL
LIN {X 0,Y 184.012,Z 449.556,A -85,B 0,C 180,E1 -24313.466,E2 -24313.466} C_VEL
LIN {X 0,Y 187.255,Z 454.503,A -85,B 0,C 180,E1 -24316.28,E2 -24316.28} C_VEL
LIN {X 0,Y 191.082,Z 460.66,A -85,B 0,C 180,E1 -24319.175,E2 -24319.175} C_VEL
LIN {X 0,Y 196.519,Z 470.021,A -85,B 0,C 180,E1 -24322.679,E2 -24322.679} C_VEL
LIN {X 0,Y 199.316,Z 475.553,A -85,B 0,C 180,E1 -24324.331,E2 -24324.331} C_VEL
LIN {X 0,Y 196.934,Z 502.327,A -85,B 0,C 180,E1 -24325.187,E2 -24325.187} C_VEL
LIN {X 0,Y 194.695,Z 515.959,A -85,B 0,C 180,E1 -24325.969,E2 -24325.969} C_VEL
LIN {X 0,Y 191.725,Z 528.02,A -85,B 0,C 180,E1 -24326.976,E2 -24326.976} C_VEL
LIN {X 0,Y 187.775,Z 540.259,A -85,B 0,C 180,E1 -24328.414,E2 -24328.414} C_VEL
LIN {X 0,Y 183.145,Z 551.718,A -85,B 0,C 180,E1 -24330.208,E2 -24330.208} C_VEL
LIN {X 0,Y 177.858,Z 562.263,A -85,B 0,C 180,E1 -24332.37,E2 -24332.37} C_VEL
LIN {X 0,Y 172.871,Z 570.884,A -85,B 0,C 180,E1 -24334.693,E2 -24334.693} C_VEL
LIN {X 0,Y 166.868,Z 579.848,A -85,B 0,C 180,E1 -24337.845,E2 -24337.845} C_VEL
LIN {X 0,Y 161.522,Z 586.779,A -85,B 0,C 180,E1 -24341.14,E2 -24341.14} C_VEL
LIN {X 0,Y 157.112,Z 591.85,A -85,B 0,C 180,E1 -24344.299,E2 -24344.299} C_VEL
LIN {X 0,Y 152.626,Z 596.446,A -85,B 0,C 180,E1 -24348.171,E2 -24348.171} C_VEL
LIN {X 0,Y 148.875,Z 599.778,A -85,B 0,C 180,E1 -24352.144,E2 -24352.144} C_VEL
LIN {X 0,Y 146.768,Z 601.42,A -85,B 0,C 180,E1 -24354.928,E2 -24354.928} C_VEL
LIN {X 0,Y 144.964,Z 602.627,A -85,B 0,C 180,E1 -24357.773,E2 -24357.773} C_VEL
LIN {X 0,Y 142.789,Z 603.597,A -85,B 0,C 180,E1 -24362.371,E2 -24362.371} C_VEL
LIN {X 0,Y 141.392,Z 603.547,A -85,B 0,C 180,E1 -24366.57,E2 -24366.57} C_VEL
LIN {X 0,Y 140.55,Z 602.299,A -85,B 0,C 180,E1 -24371.821,E2 -24371.821} C_VEL
LIN {X 0,Y 140.415,Z 600.617,A -85,B 0,C 180,E1 -24375.508,E2 -24375.508} C_VEL
LIN {X 0,Y 140.81,Z 597.681,A -85,B 0,C 180,E1 -24379.94,E2 -24379.94} C_VEL
LIN {X 0,Y 141.739,Z 593.689,A -85,B 0,C 180,E1 -24384.309,E2 -24384.309} C_VEL
LIN {X 0,Y 143.115,Z 588.554,A -85,B 0,C 180,E1 -24388.593,E2 -24388.593} C_VEL
LIN {X 0,Y 144.963,Z 582.11,A -85,B 0,C 180,E1 -24392.779,E2 -24392.779} C_VEL
LIN {X 0,Y 147.501,Z 574.026,A -85,B 0,C 180,E1 -24396.841,E2 -24396.841} C_VEL
LIN {X 0,Y 150.163,Z 565.266,A -85,B 0,C 180,E1 -24400.311,E2 -24400.311} C_VEL
LIN {X 0,Y 152.919,Z 555.762,A -85,B 0,C 180,E1 -24403.285,E2 -24403.285} C_VEL
LIN {X 0,Y 155.537,Z 545.829,A -85,B 0,C 180,E1 -24405.73,E2 -24405.73} C_VEL
LIN {X 0,Y 158.388,Z 533.254,A -85,B 0,C 180,E1 -24408.095,E2 -24408.095} C_VEL
LIN {X 0,Y 160.613,Z 520.9,A -85,B 0,C 180,E1 -24409.823,E2 -24409.823} C_VEL
LIN {X 0,Y 162.346,Z 507.723,A -85,B 0,C 180,E1 -24411.096,E2 -24411.096} C_VEL
LIN {X 0,Y 163.426,Z 494.31,A -85,B 0,C 180,E1 -24411.911,E2 -24411.911} C_VEL
LIN {X 0,Y 166.226,Z 447.068,A -85,B 0,C 180,E1 -24413.737,E2 -24413.737} C_VEL
LIN {X 0,Y 162.311,Z 437.76,A -85,B 0,C 180,E1 -24415.158,E2 -24415.158} C_VEL
LIN {X 0,Y 156.029,Z 425.37,A -85,B 0,C 180,E1 -24417.492,E2 -24417.492} C_VEL
LIN {X 0,Y 150.195,Z 415.473,A -85,B 0,C 180,E1 -24419.8,E2 -24419.8} C_VEL
LIN {X 0,Y 147.077,Z 410.742,A -85,B 0,C 180,E1 -24421.107,E2 -24421.107} C_VEL
LIN {X 0,Y 145.428,Z 407.989,A -85,B 0,C 180,E1 -24421.848,E2 -24421.848} C_VEL
LIN {X 0,Y 143.782,Z 405.763,A -85,B 0,C 180,E1 -24422.579,E2 -24422.579} C_VEL
LIN {X 0,Y 143.168,Z 403.647,A -85,B 0,C 180,E1 -24422.985,E2 -24422.985} C_VEL
LIN {X 0,Y 143.082,Z 403.66,A -85,B 0,C 180,E1 -24428.195,E2 -24428.195} C_VEL
LIN {X 0,Y 143.056,Z 403.662,A -85,B 0,C 180,E1 -24433.454,E2 -24433.454} C_VEL
LIN {X 0,Y 143.039,Z 403.656,A -85,B 0,C 180,E1 -24437.475,E2 -24437.475} C_VEL
LIN {X 0,Y 143.075,Z 403.654,A -85,B 0,C 180,E1 -24441.806,E2 -24441.806} C_VEL
LIN {X 0,Y 143.181,Z 403.647,A -85,B 0,C 180,E1 -24447.32,E2 -24447.32} C_VEL
LIN {X 0,Y 143.188,Z 403.647,A -85,B 0,C 180,E1 -24452.063,E2 -24452.063} C_VEL
LIN {X 0,Y 143.275,Z 403.634,A -85,B 0,C 180,E1 -24458.745,E2 -24458.745} C_VEL
LIN {X 0,Y 143.293,Z 403.621,A -85,B 0,C 180,E1 -24462.885,E2 -24462.885} C_VEL
LIN {X 0,Y 143.535,Z 403.599,A -85,B 0,C 180,E1 -24468.705,E2 -24468.705} C_VEL
LIN {X 0,Y 143.625,Z 403.581,A -85,B 0,C 180,E1 -24471.558,E2 -24471.558} C_VEL
LIN {X 0,Y 144.172,Z 403.478,A -85,B 0,C 180,E1 -24479.999,E2 -24479.999} C_VEL
LIN {X 0,Y 143.622,Z 403.595,A -85,B 0,C 180,E1 -24488.441,E2 -24488.441} C_VEL
LIN {X 0,Y 143.502,Z 403.598,A -85,B 0,C 180,E1 -24491.628,E2 -24491.628} C_VEL
LIN {X 0,Y 143.297,Z 403.628,A -85,B 0,C 180,E1 -24497.113,E2 -24497.113} C_VEL
LIN {X 0,Y 143.274,Z 403.638,A -85,B 0,C 180,E1 -24501.254,E2 -24501.254} C_VEL
LIN {X 0,Y 143.188,Z 403.645,A -85,B 0,C 180,E1 -24507.937,E2 -24507.937} C_VEL
LIN {X 0,Y 143.166,Z 403.656,A -85,B 0,C 180,E1 -24513.436,E2 -24513.436} C_VEL
LIN {X 0,Y 143.122,Z 403.665,A -85,B 0,C 180,E1 -24519.669,E2 -24519.669} C_VEL
LIN {X 0,Y 143.197,Z 403.817,A -85,B 0,C 180,E1 -24520.405,E2 -24520.405} C_VEL
LIN {X 0,Y 144.152,Z 406.434,A -85,B 0,C 180,E1 -24520.928,E2 -24520.928} C_VEL
LIN {X 0,Y 146.19,Z 409.031,A -85,B 0,C 180,E1 -24521.812,E2 -24521.812} C_VEL
LIN {X 0,Y 149.385,Z 414.946,A -85,B 0,C 180,E1 -24523.244,E2 -24523.244} C_VEL
LIN {X 0,Y 154.53,Z 425.388,A -85,B 0,C 180,E1 -24525.423,E2 -24525.423} C_VEL
LIN {X 0,Y 160.117,Z 439.184,A -85,B 0,C 180,E1 -24527.703,E2 -24527.703} C_VEL
LIN {X 0,Y 163.434,Z 449.229,A -85,B 0,C 180,E1 -24529.059,E2 -24529.059} C_VEL
LIN {X 0,Y 165.023,Z 470.89,A -85,B 0,C 180,E1 -24530.559,E2 -24530.559} C_VEL
LIN {X 0,Y 162.696,Z 512.214,A -85,B 0,C 180,E1 -24532.241,E2 -24532.241} C_VEL
LIN {X 0,Y 161.299,Z 525.398,A -85,B 0,C 180,E1 -24533.195,E2 -24533.195} C_VEL
LIN {X 0,Y 159.211,Z 538.315,A -85,B 0,C 180,E1 -24534.595,E2 -24534.595} C_VEL
LIN {X 0,Y 157.188,Z 548.008,A -85,B 0,C 180,E1 -24536.022,E2 -24536.022} C_VEL
LIN {X 0,Y 154.403,Z 558.848,A -85,B 0,C 180,E1 -24538.054,E2 -24538.054} C_VEL
LIN {X 0,Y 152.066,Z 567.706,A -85,B 0,C 180,E1 -24540.21,E2 -24540.21} C_VEL
LIN {X 0,Y 149.607,Z 576.163,A -85,B 0,C 180,E1 -24542.742,E2 -24542.742} C_VEL
LIN {X 0,Y 146.667,Z 585.344,A -85,B 0,C 180,E1 -24546.166,E2 -24546.166} C_VEL
LIN {X 0,Y 144.414,Z 593.45,A -85,B 0,C 180,E1 -24550.083,E2 -24550.083} C_VEL
LIN {X 0,Y 142.485,Z 600.265,A -85,B 0,C 180,E1 -24554.26,E2 -24554.26} C_VEL
LIN {X 0,Y 141.374,Z 605.703,A -85,B 0,C 180,E1 -24558.531,E2 -24558.531} C_VEL
LIN {X 0,Y 140.877,Z 609.92,A -85,B 0,C 180,E1 -24562.836,E2 -24562.836} C_VEL
LIN {X 0,Y 140.803,Z 613.03,A -85,B 0,C 180,E1 -24567.139,E2 -24567.139} C_VEL
LIN {X 0,Y 140.985,Z 614.561,A -85,B 0,C 180,E1 -24570,E2 -24570} C_VEL
LIN {X 0,Y 140.727,Z 616.046,A -85,B 0,C 180,E1 -24574.867,E2 -24574.867} C_VEL
LIN {X 0,Y 140.148,Z 616.397,A -85,B 0,C 180,E1 -24577.257,E2 -24577.257} C_VEL
LIN {X 0,Y 137.805,Z 616.231,A -85,B 0,C 180,E1 -24581.227,E2 -24581.227} C_VEL
LIN {X 0,Y 136.208,Z 615.689,A -85,B 0,C 180,E1 -24584.488,E2 -24584.488} C_VEL
LIN {X 0,Y 136.073,Z 615.026,A -85,B 0,C 180,E1 -24586.973,E2 -24586.973} C_VEL
LIN {X 0,Y 136.349,Z 614.751,A -85,B 0,C 180,E1 -24587.791,E2 -24587.791} C_VEL
LIN {X 0,Y 138.127,Z 613.415,A -85,B 0,C 180,E1 -24590.864,E2 -24590.864} C_VEL
LIN {X 0,Y 142.464,Z 609.683,A -85,B 0,C 180,E1 -24596.358,E2 -24596.358} C_VEL
LIN {X 0,Y 146.478,Z 605.685,A -85,B 0,C 180,E1 -24600.273,E2 -24600.273} C_VEL
LIN {X 0,Y 151.13,Z 600.634,A -85,B 0,C 180,E1 -24603.919,E2 -24603.919} C_VEL
LIN {X 0,Y 156.506,Z 594.308,A -85,B 0,C 180,E1 -24607.316,E2 -24607.316} C_VEL
LIN {X 0,Y 162.479,Z 586.43,A -85,B 0,C 180,E1 -24610.452,E2 -24610.452} C_VEL
LIN {X 0,Y 169.032,Z 576.658,A -85,B 0,C 180,E1 -24613.316,E2 -24613.316} C_VEL
LIN {X 0,Y 174.174,Z 567.656,A -85,B 0,C 180,E1 -24615.329,E2 -24615.329} C_VEL
LIN {X 0,Y 179.653,Z 556.531,A -85,B 0,C 180,E1 -24617.179,E2 -24617.179} C_VEL
LIN {X 0,Y 184.648,Z 543.93,A -85,B 0,C 180,E1 -24618.738,E2 -24618.738} C_VEL
LIN {X 0,Y 188.553,Z 531.078,A -85,B 0,C 180,E1 -24619.874,E2 -24619.874} C_VEL
LIN {X 0,Y 191.258,Z 518.853,A -85,B 0,C 180,E1 -24620.615,E2 -24620.615} C_VEL
LIN {X 0,Y 193.096,Z 505.086,A -85,B 0,C 180,E1 -24621.177,E2 -24621.177} C_VEL
LIN {X 0,Y 194.473,Z 487.345,A -85,B 0,C 180,E1 -24621.767,E2 -24621.767} C_VEL
LIN {X 0,Y 190.887,Z 477.661,A -85,B 0,C 180,E1 -24624.288,E2 -24624.288} C_VEL
LIN {X 0,Y 186.688,Z 468.21,A -85,B 0,C 180,E1 -24627.53,E2 -24627.53} C_VEL
LIN {X 0,Y 183.434,Z 461.475,A -85,B 0,C 180,E1 -24630.426,E2 -24630.426} C_VEL
LIN {X 0,Y 181.239,Z 457.286,A -85,B 0,C 180,E1 -24632.626,E2 -24632.626} C_VEL
LIN {X 0,Y 178.62,Z 452.303,A -85,B 0,C 180,E1 -24635.676,E2 -24635.676} C_VEL
LIN {X 0,Y 176.004,Z 447.501,A -85,B 0,C 180,E1 -24639.487,E2 -24639.487} C_VEL
LIN {X 0,Y 174.21,Z 445.039,A -85,B 0,C 180,E1 -24642.918,E2 -24642.918} C_VEL
LIN {X 0,Y 172.698,Z 441.332,A -85,B 0,C 180,E1 -24648.26,E2 -24648.26} C_VEL
LIN {X 0,Y 172.491,Z 441.213,A -85,B 0,C 180,E1 -24655.326,E2 -24655.326} C_VEL
LIN {X 0,Y 173.046,Z 441.479,A -85,B 0,C 180,E1 -24657.818,E2 -24657.818} C_VEL
LIN {X 0,Y 174.112,Z 444.542,A -85,B 0,C 180,E1 -24661.446,E2 -24661.446} C_VEL
LIN {X 0,Y 176.089,Z 446.635,A -85,B 0,C 180,E1 -24665.153,E2 -24665.153} C_VEL
LIN {X 0,Y 178.264,Z 450.245,A -85,B 0,C 180,E1 -24668.36,E2 -24668.36} C_VEL
LIN {X 0,Y 179.342,Z 451.707,A -85,B 0,C 180,E1 -24669.659,E2 -24669.659} C_VEL
LIN {X 0,Y 182.211,Z 456.035,A -85,B 0,C 180,E1 -24672.729,E2 -24672.729} C_VEL
LIN {X 0,Y 185.001,Z 460.422,A -85,B 0,C 180,E1 -24675.292,E2 -24675.292} C_VEL
LIN {X 0,Y 188.694,Z 466.605,A -85,B 0,C 180,E1 -24678.262,E2 -24678.262} C_VEL
LIN {X 0,Y 193.634,Z 475.544,A -85,B 0,C 180,E1 -24681.666,E2 -24681.666} C_VEL
LIN {X 0,Y 195.236,Z 478.99,A -85,B 0,C 180,E1 -24682.698,E2 -24682.698} C_VEL
LIN {X 0,Y 192.986,Z 503.01,A -85,B 0,C 180,E1 -24683.474,E2 -24683.474} C_VEL
LIN {X 0,Y 190.664,Z 516.527,A -85,B 0,C 180,E1 -24684.249,E2 -24684.249} C_VEL
LIN {X 0,Y 187.476,Z 528.829,A -85,B 0,C 180,E1 -24685.274,E2 -24685.274} C_VEL
LIN {X 0,Y 183.707,Z 540.112,A -85,B 0,C 180,E1 -24686.591,E2 -24686.591} C_VEL
LIN {X 0,Y 179.316,Z 550.717,A -85,B 0,C 180,E1 -24688.214,E2 -24688.214} C_VEL
LIN {X 0,Y 173.98,Z 561.28,A -85,B 0,C 180,E1 -24690.296,E2 -24690.296} C_VEL
LIN {X 0,Y 167.995,Z 571.246,A -85,B 0,C 180,E1 -24692.947,E2 -24692.947} C_VEL
LIN {X 0,Y 162.381,Z 579.28,A -85,B 0,C 180,E1 -24695.758,E2 -24695.758} C_VEL
LIN {X 0,Y 157.183,Z 585.82,A -85,B 0,C 180,E1 -24698.755,E2 -24698.755} C_VEL
LIN {X 0,Y 151.973,Z 591.629,A -85,B 0,C 180,E1 -24702.277,E2 -24702.277} C_VEL
LIN {X 0,Y 146.846,Z 596.599,A -85,B 0,C 180,E1 -24706.456,E2 -24706.456} C_VEL
LIN {X 0,Y 143.024,Z 599.824,A -85,B 0,C 180,E1 -24710.299,E2 -24710.299} C_VEL
LIN {X 0,Y 140.687,Z 601.523,A -85,B 0,C 180,E1 -24713.17,E2 -24713.17} C_VEL
LIN {X 0,Y 138.664,Z 602.789,A -85,B 0,C 180,E1 -24716.117,E2 -24716.117} C_VEL
LIN {X 0,Y 135.961,Z 603.944,A -85,B 0,C 180,E1 -24721.494,E2 -24721.494} C_VEL
LIN {X 0,Y 134.596,Z 603.923,A -85,B 0,C 180,E1 -24725.31,E2 -24725.31} C_VEL
LIN {X 0,Y 133.874,Z 603.466,A -85,B 0,C 180,E1 -24728.44,E2 -24728.44} C_VEL
LIN {X 0,Y 133.471,Z 602.548,A -85,B 0,C 180,E1 -24731.583,E2 -24731.583} C_VEL
LIN {X 0,Y 133.326,Z 601.208,A -85,B 0,C 180,E1 -24734.719,E2 -24734.719} C_VEL
LIN {X 0,Y 133.618,Z 598.386,A -85,B 0,C 180,E1 -24739.392,E2 -24739.392} C_VEL
LIN {X 0,Y 134.539,Z 594.51,A -85,B 0,C 180,E1 -24744.003,E2 -24744.003} C_VEL
LIN {X 0,Y 135.902,Z 589.504,A -85,B 0,C 180,E1 -24748.518,E2 -24748.518} C_VEL
LIN {X 0,Y 137.808,Z 583.217,A -85,B 0,C 180,E1 -24752.923,E2 -24752.923} C_VEL
LIN {X 0,Y 140.375,Z 575.363,A -85,B 0,C 180,E1 -24757.19,E2 -24757.19} C_VEL
LIN {X 0,Y 143.532,Z 565.529,A -85,B 0,C 180,E1 -24761.295,E2 -24761.295} C_VEL
LIN {X 0,Y 146.307,Z 556.446,A -85,B 0,C 180,E1 -24764.251,E2 -24764.251} C_VEL
LIN {X 0,Y 149.398,Z 545.192,A -85,B 0,C 180,E1 -24767.098,E2 -24767.098} C_VEL
LIN {X 0,Y 152.032,Z 534.151,A -85,B 0,C 180,E1 -24769.23,E2 -24769.23} C_VEL
LIN {X 0,Y 154.346,Z 521.974,A -85,B 0,C 180,E1 -24771.013,E2 -24771.013} C_VEL
LIN {X 0,Y 156.121,Z 509.626,A -85,B 0,C 180,E1 -24772.288,E2 -24772.288} C_VEL
LIN {X 0,Y 157.354,Z 495.6,A -85,B 0,C 180,E1 -24773.205,E2 -24773.205} C_VEL
LIN {X 0,Y 160.183,Z 448.551,A -85,B 0,C 180,E1 -24775.101,E2 -24775.101} C_VEL
LIN {X 0,Y 154.913,Z 436.845,A -85,B 0,C 180,E1 -24777.136,E2 -24777.136} C_VEL
LIN {X 0,Y 147.997,Z 423.778,A -85,B 0,C 180,E1 -24779.975,E2 -24779.975} C_VEL
LIN {X 0,Y 141.253,Z 413.07,A -85,B 0,C 180,E1 -24783.006,E2 -24783.006} C_VEL
LIN {X 0,Y 139.116,Z 409.667,A -85,B 0,C 180,E1 -24784.061,E2 -24784.061} C_VEL
LIN {X 0,Y 136.806,Z 406.985,A -85,B 0,C 180,E1 -24785.186,E2 -24785.186} C_VEL
LIN {X 0,Y 136.052,Z 404.533,A -85,B 0,C 180,E1 -24785.776,E2 -24785.776} C_VEL
LIN {X 0,Y 136.034,Z 404.539,A -85,B 0,C 180,E1 -24789.198,E2 -24789.198} C_VEL
LIN {X 0,Y 135.997,Z 404.542,A -85,B 0,C 180,E1 -24793.655,E2 -24793.655} C_VEL
LIN {X 0,Y 135.984,Z 404.536,A -85,B 0,C 180,E1 -24797.787,E2 -24797.787} C_VEL
LIN {X 0,Y 136.024,Z 404.532,A -85,B 0,C 180,E1 -24801.682,E2 -24801.682} C_VEL
LIN {X 0,Y 136.084,Z 404.533,A -85,B 0,C 180,E1 -24805.72,E2 -24805.72} C_VEL
LIN {X 0,Y 136.144,Z 404.525,A -85,B 0,C 180,E1 -24812.315,E2 -24812.315} C_VEL
LIN {X 0,Y 136.242,Z 404.51,A -85,B 0,C 180,E1 -24818.832,E2 -24818.832} C_VEL
LIN {X 0,Y 136.261,Z 404.501,A -85,B 0,C 180,E1 -24825.054,E2 -24825.054} C_VEL
LIN {X 0,Y 136.429,Z 404.487,A -85,B 0,C 180,E1 -24828.165,E2 -24828.165} C_VEL
LIN {X 0,Y 136.55,Z 404.46,A -85,B 0,C 180,E1 -24831.117,E2 -24831.117} C_VEL
LIN {X 0,Y 137.129,Z 404.354,A -85,B 0,C 180,E1 -24839.999,E2 -24839.999} C_VEL
LIN {X 0,Y 136.548,Z 404.475,A -85,B 0,C 180,E1 -24848.882,E2 -24848.882} C_VEL
LIN {X 0,Y 136.438,Z 404.478,A -85,B 0,C 180,E1 -24851.89,E2 -24851.89} C_VEL
LIN {X 0,Y 136.238,Z 404.504,A -85,B 0,C 180,E1 -24858.029,E2 -24858.029} C_VEL
LIN {X 0,Y 136.195,Z 404.52,A -85,B 0,C 180,E1 -24861.748,E2 -24861.748} C_VEL
LIN {X 0,Y 136.098,Z 404.529,A -85,B 0,C 180,E1 -24868.616,E2 -24868.616} C_VEL
LIN {X 0,Y 136.08,Z 404.54,A -85,B 0,C 180,E1 -24874.618,E2 -24874.618} C_VEL
LIN {X 0,Y 136.068,Z 404.544,A -85,B 0,C 180,E1 -24877.656,E2 -24877.656} C_VEL
LIN {X 0,Y 136.999,Z 407.232,A -85,B 0,C 180,E1 -24878.246,E2 -24878.246} C_VEL
LIN {X 0,Y 139.266,Z 409.968,A -85,B 0,C 180,E1 -24879.348,E2 -24879.348} C_VEL
LIN {X 0,Y 141.44,Z 413.305,A -85,B 0,C 180,E1 -24880.409,E2 -24880.409} C_VEL
LIN {X 0,Y 144.86,Z 419.434,A -85,B 0,C 180,E1 -24882.037,E2 -24882.037} C_VEL
LIN {X 0,Y 150.595,Z 431.612,A -85,B 0,C 180,E1 -24884.644,E2 -24884.644} C_VEL
LIN {X 0,Y 155.552,Z 444.803,A -85,B 0,C 180,E1 -24886.828,E2 -24886.828} C_VEL
LIN {X 0,Y 157.679,Z 451.058,A -85,B 0,C 180,E1 -24887.739,E2 -24887.739} C_VEL
LIN {X 0,Y 159.054,Z 471.787,A -85,B 0,C 180,E1 -24889.22,E2 -24889.22} C_VEL
LIN {X 0,Y 156.649,Z 512.293,A -85,B 0,C 180,E1 -24890.92,E2 -24890.92} C_VEL
LIN {X 0,Y 155.059,Z 526.111,A -85,B 0,C 180,E1 -24891.967,E2 -24891.967} C_VEL
LIN {X 0,Y 152.998,Z 538.192,A -85,B 0,C 180,E1 -24893.334,E2 -24893.334} C_VEL
LIN {X 0,Y 150.895,Z 547.842,A -85,B 0,C 180,E1 -24894.805,E2 -24894.805} C_VEL
LIN {X 0,Y 147.999,Z 558.65,A -85,B 0,C 180,E1 -24896.901,E2 -24896.901} C_VEL
LIN {X 0,Y 145.859,Z 566.287,A -85,B 0,C 180,E1 -24898.804,E2 -24898.804} C_VEL
LIN {X 0,Y 143.252,Z 574.927,A -85,B 0,C 180,E1 -24901.424,E2 -24901.424} C_VEL
LIN {X 0,Y 139.982,Z 584.738,A -85,B 0,C 180,E1 -24905.173,E2 -24905.173} C_VEL
LIN {X 0,Y 137.703,Z 592.55,A -85,B 0,C 180,E1 -24909.068,E2 -24909.068} C_VEL
LIN {X 0,Y 135.611,Z 599.468,A -85,B 0,C 180,E1 -24913.439,E2 -24913.439} C_VEL
LIN {X 0,Y 134.393,Z 605,A -85,B 0,C 180,E1 -24917.926,E2 -24917.926} C_VEL
LIN {X 0,Y 133.812,Z 609.303,A -85,B 0,C 180,E1 -24922.455,E2 -24922.455} C_VEL
LIN {X 0,Y 133.716,Z 612.493,A -85,B 0,C 180,E1 -24926.987,E2 -24926.987} C_VEL
LIN {X 0,Y 133.888,Z 614.062,A -85,B 0,C 180,E1 -24930,E2 -24930} C_VEL
LIN {X 0,Y 133.65,Z 615.588,A -85,B 0,C 180,E1 -24934.888,E2 -24934.888} C_VEL
LIN {X 0,Y 133.867,Z 616.122,A -85,B 0,C 180,E1 -24939.062,E2 -24939.062} C_VEL
LIN {X 0,Y 135.266,Z 615.562,A -85,B 0,C 180,E1 -24945.057,E2 -24945.057} C_VEL
LIN {X 0,Y 136.349,Z 614.751,A -85,B 0,C 180,E1 -24947.791,E2 -24947.791} C_VEL
LIN {X 0,Y 136.962,Z 613.893,A -85,B 0,C 180,E1 -24950.234,E2 -24950.234} C_VEL
LIN {X 0,Y 136.855,Z 611.9,A -85,B 0,C 180,E1 -24954.306,E2 -24954.306} C_VEL
LIN {X 0,Y 137.122,Z 609.752,A -85,B 0,C 180,E1 -24957.506,E2 -24957.506} C_VEL
LIN {X 0,Y 138.29,Z 607.782,A -85,B 0,C 180,E1 -24959.778,E2 -24959.778} C_VEL
LIN {X 0,Y 138.956,Z 607.057,A -85,B 0,C 180,E1 -24960.485,E2 -24960.485} C_VEL
LIN {X 0,Y 143.565,Z 602.543,A -85,B 0,C 180,E1 -24964.26,E2 -24964.26} C_VEL
LIN {X 0,Y 149.948,Z 595.631,A -85,B 0,C 180,E1 -24968.39,E2 -24968.39} C_VEL
LIN {X 0,Y 156.101,Z 588.185,A -85,B 0,C 180,E1 -24971.61,E2 -24971.61} C_VEL
LIN {X 0,Y 161.641,Z 580.624,A -85,B 0,C 180,E1 -24974.079,E2 -24974.079} C_VEL
LIN {X 0,Y 167.438,Z 571.506,A -85,B 0,C 180,E1 -24976.388,E2 -24976.388} C_VEL
LIN {X 0,Y 173.026,Z 561.401,A -85,B 0,C 180,E1 -24978.274,E2 -24978.274} C_VEL
LIN {X 0,Y 178.146,Z 550.227,A -85,B 0,C 180,E1 -24979.848,E2 -24979.848} C_VEL
LIN {X 0,Y 182.549,Z 538.181,A -85,B 0,C 180,E1 -24981.122,E2 -24981.122} C_VEL
LIN {X 0,Y 186.06,Z 525.418,A -85,B 0,C 180,E1 -24982.08,E2 -24982.08} C_VEL
LIN {X 0,Y 188.515,Z 512.503,A -85,B 0,C 180,E1 -24982.714,E2 -24982.714} C_VEL
LIN {X 0,Y 190.656,Z 490.239,A -85,B 0,C 180,E1 -24983.452,E2 -24983.452} C_VEL
LIN {X 0,Y 187.395,Z 481.362,A -85,B 0,C 180,E1 -24985.952,E2 -24985.952} C_VEL
LIN {X 0,Y 183.704,Z 472.508,A -85,B 0,C 180,E1 -24989.137,E2 -24989.137} C_VEL
LIN {X 0,Y 180.88,Z 466.581,A -85,B 0,C 180,E1 -24991.885,E2 -24991.885} C_VEL
LIN {X 0,Y 179.2,Z 463.189,A -85,B 0,C 180,E1 -24993.726,E2 -24993.726} C_VEL
LIN {X 0,Y 176.989,Z 458.743,A -85,B 0,C 180,E1 -24996.507,E2 -24996.507} C_VEL
LIN {X 0,Y 174.559,Z 454.029,A -85,B 0,C 180,E1 -25000.369,E2 -25000.369} C_VEL
LIN {X 0,Y 172.865,Z 451.508,A -85,B 0,C 180,E1 -25003.993,E2 -25003.993} C_VEL
LIN {X 0,Y 171.691,Z 448.332,A -85,B 0,C 180,E1 -25008.856,E2 -25008.856} C_VEL
LIN {X 0,Y 172.002,Z 448.359,A -85,B 0,C 180,E1 -25017.2,E2 -25017.2} C_VEL
LIN {X 0,Y 173.209,Z 451.673,A -85,B 0,C 180,E1 -25021.454,E2 -25021.454} C_VEL
LIN {X 0,Y 174.828,Z 453.513,A -85,B 0,C 180,E1 -25024.612,E2 -25024.612} C_VEL
LIN {X 0,Y 177.129,Z 457.266,A -85,B 0,C 180,E1 -25028.127,E2 -25028.127} C_VEL
LIN {X 0,Y 180.335,Z 462.319,A -85,B 0,C 180,E1 -25031.863,E2 -25031.863} C_VEL
LIN {X 0,Y 183.145,Z 466.96,A -85,B 0,C 180,E1 -25034.597,E2 -25034.597} C_VEL
LIN {X 0,Y 186.534,Z 472.932,A -85,B 0,C 180,E1 -25037.473,E2 -25037.473} C_VEL
LIN {X 0,Y 190.875,Z 481.176,A -85,B 0,C 180,E1 -25040.665,E2 -25040.665} C_VEL
LIN {X 0,Y 191.262,Z 481.916,A -85,B 0,C 180,E1 -25040.925,E2 -25040.925} C_VEL
LIN {X 0,Y 189.283,Z 503.163,A -85,B 0,C 180,E1 -25041.662,E2 -25041.662} C_VEL
LIN {X 0,Y 186.832,Z 516.942,A -85,B 0,C 180,E1 -25042.439,E2 -25042.439} C_VEL
LIN {X 0,Y 183.429,Z 529.564,A -85,B 0,C 180,E1 -25043.489,E2 -25043.489} C_VEL
LIN {X 0,Y 179.193,Z 541.625,A -85,B 0,C 180,E1 -25044.913,E2 -25044.913} C_VEL
LIN {X 0,Y 174.685,Z 551.922,A -85,B 0,C 180,E1 -25046.515,E2 -25046.515} C_VEL
LIN {X 0,Y 169.116,Z 562.346,A -85,B 0,C 180,E1 -25048.613,E2 -25048.613} C_VEL
LIN {X 0,Y 163.266,Z 571.627,A -85,B 0,C 180,E1 -25051.103,E2 -25051.103} C_VEL
LIN {X 0,Y 157.03,Z 580.114,A -85,B 0,C 180,E1 -25054.11,E2 -25054.11} C_VEL
LIN {X 0,Y 150.835,Z 587.392,A -85,B 0,C 180,E1 -25057.62,E2 -25057.62} C_VEL
LIN {X 0,Y 145.22,Z 593.114,A -85,B 0,C 180,E1 -25061.4,E2 -25061.4} C_VEL
LIN {X 0,Y 140.248,Z 597.531,A -85,B 0,C 180,E1 -25065.449,E2 -25065.449} C_VEL
LIN {X 0,Y 137.351,Z 599.837,A -85,B 0,C 180,E1 -25068.305,E2 -25068.305} C_VEL
LIN {X 0,Y 134.402,Z 601.828,A -85,B 0,C 180,E1 -25071.663,E2 -25071.663} C_VEL
LIN {X 0,Y 130.629,Z 603.846,A -85,B 0,C 180,E1 -25077.453,E2 -25077.453} C_VEL
LIN {X 0,Y 129.113,Z 604.294,A -85,B 0,C 180,E1 -25080.667,E2 -25080.667} C_VEL
LIN {X 0,Y 127.895,Z 604.297,A -85,B 0,C 180,E1 -25083.922,E2 -25083.922} C_VEL
LIN {X 0,Y 126.998,Z 603.895,A -85,B 0,C 180,E1 -25087.209,E2 -25087.209} C_VEL
LIN {X 0,Y 126.447,Z 602.949,A -85,B 0,C 180,E1 -25090.89,E2 -25090.89} C_VEL
LIN {X 0,Y 126.289,Z 600.096,A -85,B 0,C 180,E1 -25097.138,E2 -25097.138} C_VEL
LIN {X 0,Y 126.974,Z 596.689,A -85,B 0,C 180,E1 -25102.048,E2 -25102.048} C_VEL
LIN {X 0,Y 128.169,Z 592.199,A -85,B 0,C 180,E1 -25106.857,E2 -25106.857} C_VEL
LIN {X 0,Y 129.918,Z 586.502,A -85,B 0,C 180,E1 -25111.55,E2 -25111.55} C_VEL
LIN {X 0,Y 132.32,Z 579.377,A -85,B 0,C 180,E1 -25116.098,E2 -25116.098} C_VEL
LIN {X 0,Y 135.386,Z 570.456,A -85,B 0,C 180,E1 -25120.469,E2 -25120.469} C_VEL
LIN {X 0,Y 138.55,Z 561.199,A -85,B 0,C 180,E1 -25123.98,E2 -25123.98} C_VEL
LIN {X 0,Y 141.487,Z 551.233,A -85,B 0,C 180,E1 -25126.967,E2 -25126.967} C_VEL
LIN {X 0,Y 144.527,Z 539.985,A -85,B 0,C 180,E1 -25129.53,E2 -25129.53} C_VEL
LIN {X 0,Y 147.331,Z 527.398,A -85,B 0,C 180,E1 -25131.696,E2 -25131.696} C_VEL
LIN {X 0,Y 149.516,Z 514.462,A -85,B 0,C 180,E1 -25133.274,E2 -25133.274} C_VEL
LIN {X 0,Y 151.079,Z 500.699,A -85,B 0,C 180,E1 -25134.384,E2 -25134.384} C_VEL
LIN {X 0,Y 154.268,Z 450.459,A -85,B 0,C 180,E1 -25136.525,E2 -25136.525} C_VEL
LIN {X 0,Y 149.073,Z 438.966,A -85,B 0,C 180,E1 -25138.695,E2 -25138.695} C_VEL
LIN {X 0,Y 142.956,Z 427.522,A -85,B 0,C 180,E1 -25141.412,E2 -25141.412} C_VEL
LIN {X 0,Y 137.163,Z 418.132,A -85,B 0,C 180,E1 -25144.225,E2 -25144.225} C_VEL
LIN {X 0,Y 134.595,Z 414.386,A -85,B 0,C 180,E1 -25145.56,E2 -25145.56} C_VEL
LIN {X 0,Y 132.41,Z 411.155,A -85,B 0,C 180,E1 -25146.761,E2 -25146.761} C_VEL
LIN {X 0,Y 131.8,Z 410.237,A -85,B 0,C 180,E1 -25147.11,E2 -25147.11} C_VEL
LIN {X 0,Y 129.859,Z 408.051,A -85,B 0,C 180,E1 -25148.195,E2 -25148.195} C_VEL
LIN {X 0,Y 128.993,Z 405.416,A -85,B 0,C 180,E1 -25148.88,E2 -25148.88} C_VEL
LIN {X 0,Y 128.916,Z 405.421,A -85,B 0,C 180,E1 -25155.129,E2 -25155.129} C_VEL
LIN {X 0,Y 128.935,Z 405.422,A -85,B 0,C 180,E1 -25159.738,E2 -25159.738} C_VEL
LIN {X 0,Y 128.98,Z 405.414,A -85,B 0,C 180,E1 -25164.817,E2 -25164.817} C_VEL
LIN {X 0,Y 129.016,Z 405.405,A -85,B 0,C 180,E1 -25170.641,E2 -25170.641} C_VEL
LIN {X 0,Y 129.027,Z 405.409,A -85,B 0,C 180,E1 -25174.166,E2 -25174.166} C_VEL
LIN {X 0,Y 129.106,Z 405.393,A -85,B 0,C 180,E1 -25177.727,E2 -25177.727} C_VEL
LIN {X 0,Y 129.149,Z 405.393,A -85,B 0,C 180,E1 -25180.942,E2 -25180.942} C_VEL
LIN {X 0,Y 129.374,Z 405.367,A -85,B 0,C 180,E1 -25187.903,E2 -25187.903} C_VEL
LIN {X 0,Y 129.473,Z 405.341,A -85,B 0,C 180,E1 -25190.627,E2 -25190.627} C_VEL
LIN {X 0,Y 130.084,Z 405.229,A -85,B 0,C 180,E1 -25199.999,E2 -25199.999} C_VEL
LIN {X 0,Y 129.471,Z 405.356,A -85,B 0,C 180,E1 -25209.371,E2 -25209.371} C_VEL
LIN {X 0,Y 129.342,Z 405.363,A -85,B 0,C 180,E1 -25212.553,E2 -25212.553} C_VEL
LIN {X 0,Y 129.15,Z 405.389,A -85,B 0,C 180,E1 -25219.056,E2 -25219.056} C_VEL
LIN {X 0,Y 129.106,Z 405.399,A -85,B 0,C 180,E1 -25222.398,E2 -25222.398} C_VEL
LIN {X 0,Y 129.033,Z 405.413,A -85,B 0,C 180,E1 -25229.373,E2 -25229.373} C_VEL
LIN {X 0,Y 129.072,Z 405.609,A -85,B 0,C 180,E1 -25234.563,E2 -25234.563} C_VEL
LIN {X 0,Y 129.987,Z 408.201,A -85,B 0,C 180,E1 -25235.22,E2 -25235.22} C_VEL
LIN {X 0,Y 132.385,Z 410.972,A -85,B 0,C 180,E1 -25236.553,E2 -25236.553} C_VEL
LIN {X 0,Y 134.396,Z 414.144,A -85,B 0,C 180,E1 -25237.674,E2 -25237.674} C_VEL
LIN {X 0,Y 135.862,Z 416.214,A -85,B 0,C 180,E1 -25238.44,E2 -25238.44} C_VEL
LIN {X 0,Y 138.636,Z 420.487,A -85,B 0,C 180,E1 -25239.852,E2 -25239.852} C_VEL
LIN {X 0,Y 143.861,Z 431.358,A -85,B 0,C 180,E1 -25242.481,E2 -25242.481} C_VEL
LIN {X 0,Y 148.546,Z 442.931,A -85,B 0,C 180,E1 -25244.717,E2 -25244.717} C_VEL
LIN {X 0,Y 151.954,Z 453.15,A -85,B 0,C 180,E1 -25246.325,E2 -25246.325} C_VEL
LIN {X 0,Y 153.153,Z 473.043,A -85,B 0,C 180,E1 -25247.806,E2 -25247.806} C_VEL
LIN {X 0,Y 150.726,Z 511.773,A -85,B 0,C 180,E1 -25249.469,E2 -25249.469} C_VEL
LIN {X 0,Y 149.141,Z 525.16,A -85,B 0,C 180,E1 -25250.495,E2 -25250.495} C_VEL
LIN {X 0,Y 146.877,Z 537.974,A -85,B 0,C 180,E1 -25251.972,E2 -25251.972} C_VEL
LIN {X 0,Y 144.677,Z 547.601,A -85,B 0,C 180,E1 -25253.483,E2 -25253.483} C_VEL
LIN {X 0,Y 141.661,Z 558.393,A -85,B 0,C 180,E1 -25255.645,E2 -25255.645} C_VEL
LIN {X 0,Y 139.412,Z 566.019,A -85,B 0,C 180,E1 -25257.615,E2 -25257.615} C_VEL
LIN {X 0,Y 136.378,Z 575.646,A -85,B 0,C 180,E1 -25260.689,E2 -25260.689} C_VEL
LIN {X 0,Y 133.21,Z 584.553,A -85,B 0,C 180,E1 -25264.292,E2 -25264.292} C_VEL
LIN {X 0,Y 130.625,Z 592.883,A -85,B 0,C 180,E1 -25268.706,E2 -25268.706} C_VEL
LIN {X 0,Y 128.499,Z 599.683,A -85,B 0,C 180,E1 -25273.314,E2 -25273.314} C_VEL
LIN {X 0,Y 127.134,Z 605.906,A -85,B 0,C 180,E1 -25278.844,E2 -25278.844} C_VEL
LIN {X 0,Y 126.648,Z 609.91,A -85,B 0,C 180,E1 -25283.628,E2 -25283.628} C_VEL
LIN {X 0,Y 126.63,Z 612.293,A -85,B 0,C 180,E1 -25287.433,E2 -25287.433} C_VEL
LIN {X 0,Y 126.793,Z 613.558,A -85,B 0,C 180,E1 -25290,E2 -25290} C_VEL
LIN {X 0,Y 126.636,Z 614.717,A -85,B 0,C 180,E1 -25293.181,E2 -25293.181} C_VEL
LIN {X 0,Y 126.615,Z 615.449,A -85,B 0,C 180,E1 -25296.374,E2 -25296.374} C_VEL
LIN {X 0,Y 127.436,Z 615.711,A -85,B 0,C 180,E1 -25302.744,E2 -25302.744} C_VEL
LIN {X 0,Y 129.682,Z 614.477,A -85,B 0,C 180,E1 -25308.975,E2 -25308.975} C_VEL
LIN {X 0,Y 133.611,Z 611.628,A -85,B 0,C 180,E1 -25314.885,E2 -25314.885} C_VEL
LIN {X 0,Y 137.482,Z 608.415,A -85,B 0,C 180,E1 -25319.053,E2 -25319.053} C_VEL
LIN {X 0,Y 138.956,Z 607.057,A -85,B 0,C 180,E1 -25320.485,E2 -25320.485} C_VEL
LIN {X 0,Y 140.693,Z 604.861,A -85,B 0,C 180,E1 -25322.614,E2 -25322.614} C_VEL
LIN {X 0,Y 142.375,Z 600.932,A -85,B 0,C 180,E1 -25326.249,E2 -25326.249} C_VEL
LIN {X 0,Y 144.488,Z 596.446,A -85,B 0,C 180,E1 -25329.667,E2 -25329.667} C_VEL
LIN {X 0,Y 146.797,Z 593.276,A -85,B 0,C 180,E1 -25331.396,E2 -25331.396} C_VEL
LIN {X 0,Y 153.105,Z 585.694,A -85,B 0,C 180,E1 -25334.427,E2 -25334.427} C_VEL
LIN {X 0,Y 160.242,Z 575.908,A -85,B 0,C 180,E1 -25337.275,E2 -25337.275} C_VEL
LIN {X 0,Y 165.851,Z 566.884,A -85,B 0,C 180,E1 -25339.239,E2 -25339.239} C_VEL
LIN {X 0,Y 171.673,Z 555.739,A -85,B 0,C 180,E1 -25341.06,E2 -25341.06} C_VEL
LIN {X 0,Y 177.012,Z 543.107,A -85,B 0,C 180,E1 -25342.566,E2 -25342.566} C_VEL
LIN {X 0,Y 180.876,Z 531.303,A -85,B 0,C 180,E1 -25343.58,E2 -25343.58} C_VEL
LIN {X 0,Y 183.94,Z 518.512,A -85,B 0,C 180,E1 -25344.324,E2 -25344.324} C_VEL
LIN {X 0,Y 185.892,Z 504.785,A -85,B 0,C 180,E1 -25344.891,E2 -25344.891} C_VEL
LIN {X 0,Y 186.925,Z 492.993,A -85,B 0,C 180,E1 -25345.265,E2 -25345.265} C_VEL
LIN {X 0,Y 184.098,Z 485.043,A -85,B 0,C 180,E1 -25347.694,E2 -25347.694} C_VEL
LIN {X 0,Y 180.8,Z 476.891,A -85,B 0,C 180,E1 -25350.84,E2 -25350.84} C_VEL
LIN {X 0,Y 177.869,Z 470.314,A -85,B 0,C 180,E1 -25354.081,E2 -25354.081} C_VEL
LIN {X 0,Y 175.397,Z 465.14,A -85,B 0,C 180,E1 -25357.359,E2 -25357.359} C_VEL
LIN {X 0,Y 173.262,Z 460.686,A -85,B 0,C 180,E1 -25361.065,E2 -25361.065} C_VEL
LIN {X 0,Y 171.579,Z 457.996,A -85,B 0,C 180,E1 -25365.088,E2 -25365.088} C_VEL
LIN {X 0,Y 170.814,Z 455.492,A -85,B 0,C 180,E1 -25368.736,E2 -25368.736} C_VEL
LIN {X 0,Y 170.714,Z 455.281,A -85,B 0,C 180,E1 -25375.278,E2 -25375.278} C_VEL
LIN {X 0,Y 171.081,Z 455.633,A -85,B 0,C 180,E1 -25377.185,E2 -25377.185} C_VEL
LIN {X 0,Y 172.181,Z 458.667,A -85,B 0,C 180,E1 -25381.17,E2 -25381.17} C_VEL
LIN {X 0,Y 173.573,Z 460.33,A -85,B 0,C 180,E1 -25384.036,E2 -25384.036} C_VEL
LIN {X 0,Y 176.237,Z 464.875,A -85,B 0,C 180,E1 -25388.24,E2 -25388.24} C_VEL
LIN {X 0,Y 178.753,Z 469.079,A -85,B 0,C 180,E1 -25391.266,E2 -25391.266} C_VEL
LIN {X 0,Y 181.665,Z 474.079,A -85,B 0,C 180,E1 -25394.215,E2 -25394.215} C_VEL
LIN {X 0,Y 185.516,Z 481.35,A -85,B 0,C 180,E1 -25397.571,E2 -25397.571} C_VEL
LIN {X 0,Y 187.55,Z 485.467,A -85,B 0,C 180,E1 -25399.163,E2 -25399.163} C_VEL
LIN {X 0,Y 185.587,Z 504.644,A -85,B 0,C 180,E1 -25399.836,E2 -25399.836} C_VEL
LIN {X 0,Y 183.222,Z 517.168,A -85,B 0,C 180,E1 -25400.536,E2 -25400.536} C_VEL
LIN {X 0,Y 179.901,Z 529.299,A -85,B 0,C 180,E1 -25401.529,E2 -25401.529} C_VEL
LIN {X 0,Y 175.502,Z 541.478,A -85,B 0,C 180,E1 -25402.925,E2 -25402.925} C_VEL
LIN {X 0,Y 170.214,Z 553.11,A -85,B 0,C 180,E1 -25404.723,E2 -25404.723} C_VEL
LIN {X 0,Y 164.4,Z 563.403,A -85,B 0,C 180,E1 -25406.827,E2 -25406.827} C_VEL
LIN {X 0,Y 158.101,Z 572.898,A -85,B 0,C 180,E1 -25409.434,E2 -25409.434} C_VEL
LIN {X 0,Y 151.825,Z 580.941,A -85,B 0,C 180,E1 -25412.352,E2 -25412.352} C_VEL
LIN {X 0,Y 145.337,Z 588.099,A -85,B 0,C 180,E1 -25415.909,E2 -25415.909} C_VEL
LIN {X 0,Y 138.499,Z 594.577,A -85,B 0,C 180,E1 -25420.435,E2 -25420.435} C_VEL
LIN {X 0,Y 133.38,Z 598.727,A -85,B 0,C 180,E1 -25424.658,E2 -25424.658} C_VEL
LIN {X 0,Y 128.087,Z 602.215,A -85,B 0,C 180,E1 -25430.191,E2 -25430.191} C_VEL
LIN {X 0,Y 124.363,Z 604.061,A -85,B 0,C 180,E1 -25435.59,E2 -25435.59} C_VEL
LIN {X 0,Y 122.419,Z 604.633,A -85,B 0,C 180,E1 -25439.447,E2 -25439.447} C_VEL
LIN {X 0,Y 120.182,Z 604.324,A -85,B 0,C 180,E1 -25445.837,E2 -25445.837} C_VEL
LIN {X 0,Y 119.439,Z 603.286,A -85,B 0,C 180,E1 -25450.303,E2 -25450.303} C_VEL
LIN {X 0,Y 119.139,Z 600.738,A -85,B 0,C 180,E1 -25456.352,E2 -25456.352} C_VEL
LIN {X 0,Y 119.75,Z 597.443,A -85,B 0,C 180,E1 -25461.563,E2 -25461.563} C_VEL
LIN {X 0,Y 120.97,Z 593.064,A -85,B 0,C 180,E1 -25466.669,E2 -25466.669} C_VEL
LIN {X 0,Y 122.756,Z 587.493,A -85,B 0,C 180,E1 -25471.64,E2 -25471.64} C_VEL
LIN {X 0,Y 125.193,Z 580.546,A -85,B 0,C 180,E1 -25476.446,E2 -25476.446} C_VEL
LIN {X 0,Y 127.809,Z 573.445,A -85,B 0,C 180,E1 -25480.295,E2 -25480.295} C_VEL
LIN {X 0,Y 131.09,Z 564.175,A -85,B 0,C 180,E1 -25484.247,E2 -25484.247} C_VEL
LIN {X 0,Y 134.258,Z 554.317,A -85,B 0,C 180,E1 -25487.517,E2 -25487.517} C_VEL
LIN {X 0,Y 137.427,Z 543.803,A -85,B 0,C 180,E1 -25490.193,E2 -25490.193} C_VEL
LIN {X 0,Y 140.333,Z 532.269,A -85,B 0,C 180,E1 -25492.449,E2 -25492.449} C_VEL
LIN {X 0,Y 142.7,Z 520.335,A -85,B 0,C 180,E1 -25494.166,E2 -25494.166} C_VEL
LIN {X 0,Y 144.539,Z 507.508,A -85,B 0,C 180,E1 -25495.468,E2 -25495.468} C_VEL
LIN {X 0,Y 145.751,Z 493.855,A -85,B 0,C 180,E1 -25496.312,E2 -25496.312} C_VEL
LIN {X 0,Y 148.499,Z 452.43,A -85,B 0,C 180,E1 -25498.042,E2 -25498.042} C_VEL
LIN {X 0,Y 142.459,Z 439.5,A -85,B 0,C 180,E1 -25500.787,E2 -25500.787} C_VEL
LIN {X 0,Y 137.536,Z 430.289,A -85,B 0,C 180,E1 -25503.204,E2 -25503.204} C_VEL
LIN {X 0,Y 131.161,Z 420.069,A -85,B 0,C 180,E1 -25506.625,E2 -25506.625} C_VEL
LIN {X 0,Y 128.539,Z 416.256,A -85,B 0,C 180,E1 -25508.158,E2 -25508.158} C_VEL
LIN {X 0,Y 125.854,Z 412.66,A -85,B 0,C 180,E1 -25509.815,E2 -25509.815} C_VEL
LIN {X 0,Y 125.065,Z 411.363,A -85,B 0,C 180,E1 -25510.348,E2 -25510.348} C_VEL
LIN {X 0,Y 122.888,Z 409.231,A -85,B 0,C 180,E1 -25511.748,E2 -25511.748} C_VEL
LIN {X 0,Y 121.901,Z 406.803,A -85,B 0,C 180,E1 -25512.551,E2 -25512.551} C_VEL
LIN {X 0,Y 121.826,Z 406.301,A -85,B 0,C 180,E1 -25512.763,E2 -25512.763} C_VEL
LIN {X 0,Y 121.864,Z 406.298,A -85,B 0,C 180,E1 -25518.564,E2 -25518.564} C_VEL
LIN {X 0,Y 121.931,Z 406.292,A -85,B 0,C 180,E1 -25524.802,E2 -25524.802} C_VEL
LIN {X 0,Y 121.928,Z 406.284,A -85,B 0,C 180,E1 -25529.836,E2 -25529.836} C_VEL
LIN {X 0,Y 121.982,Z 406.276,A -85,B 0,C 180,E1 -25536.214,E2 -25536.214} C_VEL
LIN {X 0,Y 122.043,Z 406.281,A -85,B 0,C 180,E1 -25539.786,E2 -25539.786} C_VEL
LIN {X 0,Y 122.237,Z 406.256,A -85,B 0,C 180,E1 -25546.703,E2 -25546.703} C_VEL
LIN {X 0,Y 122.405,Z 406.222,A -85,B 0,C 180,E1 -25550.081,E2 -25550.081} C_VEL
LIN {X 0,Y 122.596,Z 406.2,A -85,B 0,C 180,E1 -25556.713,E2 -25556.713} C_VEL
LIN {X 0,Y 123.038,Z 406.105,A -85,B 0,C 180,E1 -25559.999,E2 -25559.999} C_VEL
LIN {X 0,Y 122.421,Z 406.227,A -85,B 0,C 180,E1 -25566.592,E2 -25566.592} C_VEL
LIN {X 0,Y 122.32,Z 406.236,A -85,B 0,C 180,E1 -25572.385,E2 -25572.385} C_VEL
LIN {X 0,Y 122.105,Z 406.268,A -85,B 0,C 180,E1 -25576.725,E2 -25576.725} C_VEL
LIN {X 0,Y 122.021,Z 406.279,A -85,B 0,C 180,E1 -25582.85,E2 -25582.85} C_VEL
LIN {X 0,Y 121.947,Z 406.291,A -85,B 0,C 180,E1 -25587.454,E2 -25587.454} C_VEL
LIN {X 0,Y 121.914,Z 406.302,A -85,B 0,C 180,E1 -25590.736,E2 -25590.736} C_VEL
LIN {X 0,Y 122.772,Z 408.91,A -85,B 0,C 180,E1 -25591.489,E2 -25591.489} C_VEL
LIN {X 0,Y 124.791,Z 411.147,A -85,B 0,C 180,E1 -25592.824,E2 -25592.824} C_VEL
LIN {X 0,Y 125.565,Z 411.987,A -85,B 0,C 180,E1 -25593.313,E2 -25593.313} C_VEL
LIN {X 0,Y 127.78,Z 415.363,A -85,B 0,C 180,E1 -25594.737,E2 -25594.737} C_VEL
LIN {X 0,Y 129.019,Z 417.073,A -85,B 0,C 180,E1 -25595.481,E2 -25595.481} C_VEL
LIN {X 0,Y 133.985,Z 424.412,A -85,B 0,C 180,E1 -25598.272,E2 -25598.272} C_VEL
LIN {X 0,Y 139.092,Z 435.248,A -85,B 0,C 180,E1 -25601.06,E2 -25601.06} C_VEL
LIN {X 0,Y 143.425,Z 446.344,A -85,B 0,C 180,E1 -25603.315,E2 -25603.315} C_VEL
LIN {X 0,Y 146.398,Z 455.832,A -85,B 0,C 180,E1 -25604.863,E2 -25604.863} C_VEL
LIN {X 0,Y 147.351,Z 474.126,A -85,B 0,C 180,E1 -25606.273,E2 -25606.273} C_VEL
LIN {X 0,Y 144.86,Z 511.632,A -85,B 0,C 180,E1 -25607.925,E2 -25607.925} C_VEL
LIN {X 0,Y 143.207,Z 524.956,A -85,B 0,C 180,E1 -25608.976,E2 -25608.976} C_VEL
LIN {X 0,Y 140.845,Z 537.739,A -85,B 0,C 180,E1 -25610.491,E2 -25610.491} C_VEL
LIN {X 0,Y 138.543,Z 547.343,A -85,B 0,C 180,E1 -25612.044,E2 -25612.044} C_VEL
LIN {X 0,Y 135.398,Z 558.121,A -85,B 0,C 180,E1 -25614.273,E2 -25614.273} C_VEL
LIN {X 0,Y 133.031,Z 565.736,A -85,B 0,C 180,E1 -25616.31,E2 -25616.31} C_VEL
LIN {X 0,Y 130.148,Z 574.359,A -85,B 0,C 180,E1 -25619.137,E2 -25619.137} C_VEL
LIN {X 0,Y 126.895,Z 582.884,A -85,B 0,C 180,E1 -25622.618,E2 -25622.618} C_VEL
LIN {X 0,Y 124.851,Z 589.255,A -85,B 0,C 180,E1 -25625.914,E2 -25625.914} C_VEL
LIN {X 0,Y 122.348,Z 596.728,A -85,B 0,C 180,E1 -25630.714,E2 -25630.714} C_VEL
LIN {X 0,Y 120.855,Z 601.781,A -85,B 0,C 180,E1 -25634.83,E2 -25634.83} C_VEL
LIN {X 0,Y 119.904,Z 606.674,A -85,B 0,C 180,E1 -25639.873,E2 -25639.873} C_VEL
LIN {X 0,Y 119.531,Z 610.391,A -85,B 0,C 180,E1 -25644.94,E2 -25644.94} C_VEL
LIN {X 0,Y 119.712,Z 613.051,A -85,B 0,C 180,E1 -25650,E2 -25650} C_VEL
LIN {X 0,Y 119.558,Z 614.249,A -85,B 0,C 180,E1 -25653.37,E2 -25653.37} C_VEL
LIN {X 0,Y 119.547,Z 615.042,A -85,B 0,C 180,E1 -25656.752,E2 -25656.752} C_VEL
LIN {X 0,Y 120.495,Z 615.394,A -85,B 0,C 180,E1 -25663.491,E2 -25663.491} C_VEL
LIN {X 0,Y 122.966,Z 614.241,A -85,B 0,C 180,E1 -25670.055,E2 -25670.055} C_VEL
LIN {X 0,Y 124.917,Z 613.09,A -85,B 0,C 180,E1 -25673.192,E2 -25673.192} C_VEL
LIN {X 0,Y 127.176,Z 611.506,A -85,B 0,C 180,E1 -25676.237,E2 -25676.237} C_VEL
LIN {X 0,Y 131.299,Z 608.377,A -85,B 0,C 180,E1 -25680.563,E2 -25680.563} C_VEL
LIN {X 0,Y 136.017,Z 604.227,A -85,B 0,C 180,E1 -25684.636,E2 -25684.636} C_VEL
LIN {X 0,Y 142.435,Z 597.934,A -85,B 0,C 180,E1 -25688.983,E2 -25688.983} C_VEL
LIN {X 0,Y 146.797,Z 593.276,A -85,B 0,C 180,E1 -25691.396,E2 -25691.396} C_VEL
LIN {X 0,Y 149.222,Z 589.946,A -85,B 0,C 180,E1 -25693.025,E2 -25693.025} C_VEL
LIN {X 0,Y 152.063,Z 584.198,A -85,B 0,C 180,E1 -25695.915,E2 -25695.915} C_VEL
LIN {X 0,Y 154.945,Z 577.979,A -85,B 0,C 180,E1 -25698.578,E2 -25698.578} C_VEL
LIN {X 0,Y 157.336,Z 573.799,A -85,B 0,C 180,E1 -25699.829,E2 -25699.829} C_VEL
LIN {X 0,Y 163.961,Z 563.05,A -85,B 0,C 180,E1 -25701.962,E2 -25701.962} C_VEL
LIN {X 0,Y 169.395,Z 552.532,A -85,B 0,C 180,E1 -25703.497,E2 -25703.497} C_VEL
LIN {X 0,Y 174.213,Z 540.892,A -85,B 0,C 180,E1 -25704.775,E2 -25704.775} C_VEL
LIN {X 0,Y 178.42,Z 527.581,A -85,B 0,C 180,E1 -25705.81,E2 -25705.81} C_VEL
LIN {X 0,Y 181.275,Z 514.894,A -85,B 0,C 180,E1 -25706.464,E2 -25706.464} C_VEL
LIN {X 0,Y 183.107,Z 500.152,A -85,B 0,C 180,E1 -25706.973,E2 -25706.973} C_VEL
LIN {X 0,Y 183.416,Z 495.906,A -85,B 0,C 180,E1 -25707.155,E2 -25707.155} C_VEL
LIN {X 0,Y 181.025,Z 488.969,A -85,B 0,C 180,E1 -25709.439,E2 -25709.439} C_VEL
LIN {X 0,Y 178.365,Z 482.049,A -85,B 0,C 180,E1 -25712.248,E2 -25712.248} C_VEL
LIN {X 0,Y 175.88,Z 476.128,A -85,B 0,C 180,E1 -25715.272,E2 -25715.272} C_VEL
LIN {X 0,Y 173.781,Z 471.469,A -85,B 0,C 180,E1 -25718.316,E2 -25718.316} C_VEL
LIN {X 0,Y 172.008,Z 467.38,A -85,B 0,C 180,E1 -25721.732,E2 -25721.732} C_VEL
LIN {X 0,Y 169.863,Z 462.452,A -85,B 0,C 180,E1 -25729.14,E2 -25729.14} C_VEL
LIN {X 0,Y 169.952,Z 462.366,A -85,B 0,C 180,E1 -25735.979,E2 -25735.979} C_VEL
LIN {X 0,Y 170.157,Z 462.939,A -85,B 0,C 180,E1 -25737.17,E2 -25737.17} C_VEL
LIN {X 0,Y 171.273,Z 465.835,A -85,B 0,C 180,E1 -25741.176,E2 -25741.176} C_VEL
LIN {X 0,Y 172.408,Z 467.298,A -85,B 0,C 180,E1 -25743.603,E2 -25743.603} C_VEL
LIN {X 0,Y 174.867,Z 471.757,A -85,B 0,C 180,E1 -25747.719,E2 -25747.719} C_VEL
LIN {X 0,Y 177.123,Z 475.68,A -85,B 0,C 180,E1 -25750.575,E2 -25750.575} C_VEL
LIN {X 0,Y 180.119,Z 481.097,A -85,B 0,C 180,E1 -25753.759,E2 -25753.759} C_VEL
LIN {X 0,Y 184.003,Z 488.969,A -85,B 0,C 180,E1 -25757.283,E2 -25757.283} C_VEL
LIN {X 0,Y 182.204,Z 505.65,A -85,B 0,C 180,E1 -25757.907,E2 -25757.907} C_VEL
LIN {X 0,Y 179.639,Z 518.47,A -85,B 0,C 180,E1 -25758.634,E2 -25758.634} C_VEL
LIN {X 0,Y 175.873,Z 531.222,A -85,B 0,C 180,E1 -25759.686,E2 -25759.686} C_VEL
LIN {X 0,Y 171.382,Z 542.991,A -85,B 0,C 180,E1 -25761.07,E2 -25761.07} C_VEL
LIN {X 0,Y 165.88,Z 554.362,A -85,B 0,C 180,E1 -25762.856,E2 -25762.856} C_VEL
LIN {X 0,Y 159.863,Z 564.478,A -85,B 0,C 180,E1 -25764.946,E2 -25764.946} C_VEL
LIN {X 0,Y 154.363,Z 572.386,A -85,B 0,C 180,E1 -25767.084,E2 -25767.084} C_VEL
LIN {X 0,Y 147.955,Z 580.376,A -85,B 0,C 180,E1 -25769.903,E2 -25769.903} C_VEL
LIN {X 0,Y 141.814,Z 587.017,A -85,B 0,C 180,E1 -25773.035,E2 -25773.035} C_VEL
LIN {X 0,Y 135.779,Z 592.697,A -85,B 0,C 180,E1 -25776.653,E2 -25776.653} C_VEL
LIN {X 0,Y 129.984,Z 597.384,A -85,B 0,C 180,E1 -25780.805,E2 -25780.805} C_VEL
LIN {X 0,Y 126.517,Z 599.812,A -85,B 0,C 180,E1 -25783.769,E2 -25783.769} C_VEL
LIN {X 0,Y 121.874,Z 602.599,A -85,B 0,C 180,E1 -25788.562,E2 -25788.562} C_VEL
LIN {X 0,Y 118.265,Z 604.275,A -85,B 0,C 180,E1 -25793.541,E2 -25793.541} C_VEL
LIN {X 0,Y 115.701,Z 604.978,A -85,B 0,C 180,E1 -25798.257,E2 -25798.257} C_VEL
LIN {X 0,Y 113.448,Z 604.753,A -85,B 0,C 180,E1 -25804.302,E2 -25804.302} C_VEL
LIN {X 0,Y 112.399,Z 603.602,A -85,B 0,C 180,E1 -25809.707,E2 -25809.707} C_VEL
LIN {X 0,Y 112.116,Z 600.438,A -85,B 0,C 180,E1 -25817.327,E2 -25817.327} C_VEL
LIN {X 0,Y 113.1,Z 596.123,A -85,B 0,C 180,E1 -25823.856,E2 -25823.856} C_VEL
LIN {X 0,Y 114.891,Z 590.442,A -85,B 0,C 180,E1 -25830,E2 -25830} C_VEL
LIN {X 0,Y 117.138,Z 584.138,A -85,B 0,C 180,E1 -25835.163,E2 -25835.163} C_VEL
LIN {X 0,Y 120.193,Z 576.252,A -85,B 0,C 180,E1 -25840.103,E2 -25840.103} C_VEL
LIN {X 0,Y 123.681,Z 566.979,A -85,B 0,C 180,E1 -25844.544,E2 -25844.544} C_VEL
LIN {X 0,Y 126.768,Z 558.37,A -85,B 0,C 180,E1 -25847.753,E2 -25847.753} C_VEL
LIN {X 0,Y 130.335,Z 547.414,A -85,B 0,C 180,E1 -25850.93,E2 -25850.93} C_VEL
LIN {X 0,Y 133.769,Z 534.908,A -85,B 0,C 180,E1 -25853.615,E2 -25853.615} C_VEL
LIN {X 0,Y 136.463,Z 522.657,A -85,B 0,C 180,E1 -25855.551,E2 -25855.551} C_VEL
LIN {X 0,Y 138.553,Z 509.77,A -85,B 0,C 180,E1 -25856.958,E2 -25856.958} C_VEL
LIN {X 0,Y 139.938,Z 496.048,A -85,B 0,C 180,E1 -25857.896,E2 -25857.896} C_VEL
LIN {X 0,Y 142.782,Z 454.556,A -85,B 0,C 180,E1 -25859.691,E2 -25859.691} C_VEL
LIN {X 0,Y 136.953,Z 441.921,A -85,B 0,C 180,E1 -25862.6,E2 -25862.6} C_VEL
LIN {X 0,Y 132.268,Z 433.321,A -85,B 0,C 180,E1 -25865.114,E2 -25865.114} C_VEL
LIN {X 0,Y 127.199,Z 425.089,A -85,B 0,C 180,E1 -25868.077,E2 -25868.077} C_VEL
LIN {X 0,Y 124.117,Z 420.68,A -85,B 0,C 180,E1 -25870.031,E2 -25870.031} C_VEL
LIN {X 0,Y 121.611,Z 417.024,A -85,B 0,C 180,E1 -25871.756,E2 -25871.756} C_VEL
LIN {X 0,Y 119.286,Z 414.215,A -85,B 0,C 180,E1 -25873.426,E2 -25873.426} C_VEL
LIN {X 0,Y 118.321,Z 412.477,A -85,B 0,C 180,E1 -25874.215,E2 -25874.215} C_VEL
LIN {X 0,Y 116.055,Z 410.404,A -85,B 0,C 180,E1 -25875.962,E2 -25875.962} C_VEL
LIN {X 0,Y 114.928,Z 407.905,A -85,B 0,C 180,E1 -25877.051,E2 -25877.051} C_VEL
LIN {X 0,Y 114.786,Z 407.173,A -85,B 0,C 180,E1 -25877.282,E2 -25877.282} C_VEL
LIN {X 0,Y 114.794,Z 407.172,A -85,B 0,C 180,E1 -25882.738,E2 -25882.738} C_VEL
LIN {X 0,Y 114.861,Z 407.164,A -85,B 0,C 180,E1 -25888.936,E2 -25888.936} C_VEL
LIN {X 0,Y 114.946,Z 407.151,A -85,B 0,C 180,E1 -25896.506,E2 -25896.506} C_VEL
LIN {X 0,Y 115.007,Z 407.146,A -85,B 0,C 180,E1 -25902.208,E2 -25902.208} C_VEL
LIN {X 0,Y 115.254,Z 407.126,A -85,B 0,C 180,E1 -25907.326,E2 -25907.326} C_VEL
LIN {X 0,Y 115.364,Z 407.107,A -85,B 0,C 180,E1 -25913.001,E2 -25913.001} C_VEL
LIN {X 0,Y 115.989,Z 406.981,A -85,B 0,C 180,E1 -25919.999,E2 -25919.999} C_VEL
LIN {X 0,Y 115.361,Z 407.109,A -85,B 0,C 180,E1 -25926.998,E2 -25926.998} C_VEL
